// CNC/10 MessagesHandler/FB_ChannelError
FUNCTION_BLOCK FB_ChannelError
VAR_INPUT
	nChanIdx: INT;
END_VAR
VAR_OUTPUT
	Valid: BOOL := FALSE;
	/// Identification of channel error 
	ChErrorID: UDINT;
	/// Module name 
	ModuleName: STRING;
	/// Line in source file 
	Line: DINT;
	/// Multiple ID 
	MultipleID: DINT;
	/// Commandable function type 
	CmdFunctionType: DINT;
	/// Identification of the channel 
	ChannelID: DINT;
	/// Communication ID 
	CommuID: DINT;
	/// Cycle counter of CNC 
	CycleCounter: UDINT;
	/// Version name 
	VersionName: STRING;
	/// Remedy class of error 
	RemedyClass: DINT;
	/// Reaction class of error 
	ReactionClass: DINT;
	/// Body type of error 
	BodyType: UDINT;
	/// User message 
	UserMessage: STRING;
	/// Variables of error record body 
	BodyTypeEnum: UDINT;
	NcBlockNr: DINT := 0;
	ProgName: STRING := '';
	FileName: STRING := '';
	FileOffset: UDINT := 0;
	NcBlockOffset: DINT := 0;
	TokenOffset: DINT := 0;
	LogicalPathNr: DINT := 0;
	AddProgInfo: STRING := '';
	CommuMedium: DINT := 0;
	CommuType: UDINT := 0;
	CommuPartner: UDINT := 0;
	FileLine: UDINT := 0;
	ListType: DINT := 0;
	StructName: STRING := '';
	StrValue_1: STRING;
	StrValue_2: STRING;
	StrValue_3: STRING;
	StrValue_4: STRING;
	StrValue_5: STRING;
	MeaningValue_1: STRING;
	MeaningValue_2: STRING;
	MeaningValue_3: STRING;
	MeaningValue_4: STRING;
END_VAR
VAR
	/// Index of channel specific HLI area 	
	pMcError: POINTER TO MC_ERROR;
	pMcError2: POINTER TO MC_ERROR;
	SatzR: HLI_ERROR_SATZ;
	bInitialized: BOOL := FALSE;
	bClear: BOOL := FALSE;
	bUsed: ARRAY[0..CNC_EVENTS_MAXIDX] OF BOOL;
	bToCleanUp: ARRAY[0..CNC_EVENTS_MAXIDX] OF BOOL;
	LogEvent: ARRAY[0..CNC_EVENTS_MAXIDX] OF ADSLOGEVENT;
	FlankeQuit: ARRAY[0..CNC_EVENTS_MAXIDX] OF R_TRIG;
	pLog: POINTER TO ADSLOGEVENT;
	fmtStr: STRING;
	eventId: UDINT;
	i: UDINT;
	idx: UDINT := 0;
	maxWarnings: UINT;
	maxErrors: UINT;
	maxUserEvents: UINT;
	/// Gesamtzahl = Userevents und Errors 
	maxEvents: UINT;
	/// maximal index of an event 
	maxIdxEvents: UINT;
	countWarnings: UINT := 0;
	countErrors: UINT := 0;
	countUserEvents: UINT := 0;
	start_idx: UINT;
	stop_idx: UINT;
	paraPointerArray: ARRAY[0..31] OF POINTER TO UDINT;
	paraIndex: INT;
	pRumpfNcProg: POINTER TO HLI_RUMPF_NC_PROG;
	pRumpfNcProgLr: POINTER TO HLI_RUMPF_NC_PROG_LR;
	pRumpfMds: POINTER TO HLI_RUMPF_MDS;
	pRumpfKommu: POINTER TO HLI_RUMPF_KOMMU;
	pRumpfRamDisk: POINTER TO HLI_RUMPF_RAMDISK;
	pRumpfFile: POINTER TO HLI_RUMPF_FILE;
	pRumpfIntprFile: POINTER TO HLI_RUMPF_INTPR_FILE;
	pRumpfListeBinaer: POINTER TO HLI_RUMPF_LISTE_BINAER;
	pRumpfGcm: POINTER TO HLI_RUMPF_GCM;
	bTcComError: BOOL;
	bAxisErr: BOOL;
	nLogAxisId: DINT;
	
	// TC3 EventLogger
	fbADSRead : ADSREAD;
  	cnc_error_manager_mode_r : UDINT;
  	suppress_tc2_event_log_output : BOOL; 
	init : BOOL;
END_VAR
VAR CONSTANT
	XmlEventId_Rumpf: UDINT := 200;
	XmlEventId_RumpfNcProg: UDINT := 201;
	XmlEventId_RumpfNcProgLr: UDINT := 202;
	XmlEventId_RumpfMds: UDINT := 203;
	XmlEventId_RumpfKommu: UDINT := 204;
	XmlEventId_RumpfRamDisk: UDINT := 205;
	XmlEventId_RumpfFile: UDINT := 206;
	XmlEventId_RumpfIntprFile: UDINT := 207;
	XmlEventId_RumpfListeBinaer: UDINT := 208;
	XmlEventId_RumpfGcm: UDINT := 209;
	CNC_SOURCE_ID_BASE: UDINT := 551;
	CNC_USER_SOURCE_ID_BASE: UDINT := 651;
	MAX_CNC_ERRORS: UDINT := 49;
	MAX_CNC_USER_EVENTS: UDINT := 49;
	/// MAX_CNC_ERRORS + MAX_CNC_USER_EVENTS 
	MAX_CNC_EVENTS: UDINT := 98;
	/// MAX_CNC_EVENTS - 1 
	CNC_EVENTS_MAXIDX: UDINT := 97;
	ERR_BAHN_ONLINE_TRC_CALCULATION: UDINT := 50689;
	ERR_ID_REPORT_CNC_RESET: UDINT := 270076;
	ERR_ID_KIN_TRAFO_CONFIG: UDINT := 292030;
	ERR_ID_KIN_TRAFO_INIT: UDINT := 292031;
	ERR_ID_KIN_TRAFO_FORWARD: UDINT := 292032;
	ERR_ID_KIN_TRAFO_BACKWARD: UDINT := 292033;
END_VAR

(* ========================================================= *)
(*    FB: FB_ChannelError                               	 *)
(* --------------------------------------------------------- *)
(*   Desc: FB transfers CNC Errors to the Event Logger		 *)
(*   Author: ISG / TV                                        *)
(*   Date: 20.11.2018                                        *)
(*   Rev.: 1.6                                               *)
(*															 *)
(* ========================================================= *)

(* check for channel no *)
IF NOT HLI3_CheckChannelValid(nChannel := nChanIdx) THEN
	RETURN;
END_IF



// Check if TC3 EventLogger is active
fbADSRead(
	NETID:= '', 
	PORT:= 553, 
	IDXGRP:= 16#20101, 
	IDXOFFS:= 16#293, 
	LEN:= 4, 
	DESTADDR:= ADR(cnc_error_manager_mode_r ), 
	READ:= TRUE);
		
	IF NOT fbADSRead.BUSY THEN
		init := TRUE;
	END_IF
	
	IF NOT init THEN 
		RETURN;
	END_IF
			
	IF ((cnc_error_manager_mode_r AND 16#00080000) = 16#80000) THEN
		  suppress_tc2_event_log_output := TRUE;	
	END_IF


(* check for zero pointer *)
IF gpCh[nChanIdx] = 0 THEN
  RETURN;
END_IF

(* check for zero pointer, first channel is necessary for axis errors (Position controller errors) *)
IF gpCh[0] = 0 THEN
  RETURN;
END_IF

pMcError := ADR(gpCh[nChanIdx]^.mc_error);
SatzR    := pMcError^.satz_r;

IF bInitialized = FALSE THEN
  pMcError^.enable_w := TRUE;    (* enable control unit for error messages *) 
  bInitialized  := TRUE;
  maxErrors     := UDINT_TO_UINT(MAX_CNC_ERRORS / gNrCh);
  maxWarnings   := maxErrors / 5;
  maxUserEvents := UDINT_TO_UINT(MAX_CNC_USER_EVENTS / gNrCh);
  maxEvents     := maxUserEvents + maxErrors;

  maxIdxEvents := (maxEvents - 1);
  FOR i := 0 TO maxIdxEvents DO
    (* ----------------------------------------- *)
    (* initialize fixed elements of event        *)
    (* ----------------------------------------- *)
    pLog := ADR( LogEvent[i] );
    pLog^.NETID := '';      (* Local Computer *)
    pLog^.PORT:= 110;       (* Event Logger *)
    pLog^.TMOUT:= t#10s;
    pLog^.EventConfigData.Prio         := TCEVENTPRIO_IMPLICIT;
    pLog^.EventConfigData.ProgId       := 'TcEventFormatter.TcXmlFormatter';
    pLog^.EventConfigData.Flags        := TCEVENTFLAG_SRCID OR TCEVENTFLAG_LOG;
    pLog^.EventConfigData.SourceString := '';
    pLog^.EventConfigData.StreamType   := TCEVENTSTREAM_NORMAL;

    IF i < maxErrors THEN
      (* SourceID: 550 error texts, [ 551,  599] for single CNC error messages *)
      pLog^.EventConfigData.SourceId := CNC_SOURCE_ID_BASE + i + (DINT_TO_UINT(nChanIdx)*maxErrors);
    ELSE
      (* SourceID: 650 user error texts, [ 651,  699] for single CNC user error messages "ERROR[]" *)
      pLog^.EventConfigData.SourceId := CNC_USER_SOURCE_ID_BASE + i-maxErrors + (DINT_TO_UINT(nChanIdx)*maxUserEvents);
    END_IF

    FlankeQuit[i](CLK :=  pLog^.Quit);
  END_FOR
END_IF



(* -------------------------------------------------------------------------*)
(* test if events which have been reported shall be cleared again           *)
(* -------------------------------------------------------------------------*)
IF bClear THEN
  bClear := FALSE;
  countWarnings := 0;
  countErrors := 0;
  countUserEvents := 0;
  FOR i := 0 TO maxIdxEvents DO
    IF bToCleanup[i] = FALSE AND bUsed[i] THEN
      bToCleanup[i] := TRUE;
    END_IF
  END_FOR
END_IF


(* -------------------------------------------------------------------------*)
(* check for new error message                                              *)
(* -------------------------------------------------------------------------*)

(* Output for position controller errors is gpCh[0]^ *)
IF gpCh[0]^.mc_error.semaphor_rw THEN	
	SatzR := gpCh[0]^.mc_error.satz_r;		
	bAxisErr := TRUE;				
END_IF

IF (pMcError^.semaphor_rw  OR bAxisErr)  THEN

 	IF  SatzR.kopf.cnc_channel > 0 THEN 
  		IF (SatzR.kopf.cnc_channel-1 <> INT_TO_UINT(nChanIdx)) THEN	  
			bAxisErr := FALSE;		
    	RETURN;
	END_IF
  END_IF
  
  (* Initialize output variables that depend on error body type *)
  NcBlockNr      := 0;
  ProgName       := '';
  FileName       := '';
  FileOffset     := 0;
  NcBlockOffset  := 0;
  TokenOffset    := 0;
  LogicalPathNr  := 0;
  AddProgInfo    := '';

  CommuMedium    := 0;
  CommuType      := 0;
  CommuPartner   := 0;

  FileLine       := 0;
  ListType       := 0;
  StructName     := '';

  StrValue_1     := '';
  StrValue_2     := '';
  StrValue_3     := '';
  StrValue_4     := '';
  StrValue_5     := '';

  MeaningValue_1 := '';
  MeaningValue_2 := '';
  MeaningValue_3 := '';
  MeaningValue_4 := '';
  
  nLogAxisId   := 0;


  eventId := SatzR.kopf.error_id;

  (*------------------------------------------------------------------*)
  (* automatic clear old events if CNC reports reset                  *)
  (*------------------------------------------------------------------*)
  IF eventId = ERR_ID_REPORT_CNC_RESET THEN
	  	IF bAxisErr THEN 
    		gpCh[0]^.mc_error.semaphor_rw := FALSE;
			bAxisErr := FALSE;
		ELSE
			pMcError^.semaphor_rw := FALSE;		
		END_IF
	
    bClear := TRUE;
    RETURN;
  END_IF

  
  (*------------------------------------------------------------------*)
  (* TcCom: kinematic transformation, map util_error_id to error_id   *)
  (*------------------------------------------------------------------*)
  IF    eventId = ERR_ID_KIN_TRAFO_CONFIG
     OR eventId = ERR_ID_KIN_TRAFO_INIT  
     OR eventId = ERR_ID_KIN_TRAFO_FORWARD
     OR eventId = ERR_ID_KIN_TRAFO_BACKWARD
   OR eventId = ERR_BAHN_ONLINE_TRC_CALCULATION
  THEN
    eventId := SatzR.kopf.util_error_id;
    bTcComError := TRUE;
  ELSE
    bTcComError := FALSE;
  END_IF
   

  (*-------------------------------*)
  (* search unused event           *)
  (*-------------------------------*)
  IF eventId <= 1000 OR bTcComError THEN
    countUserEvents := countUserEvents + 1;
    start_idx       := maxErrors;
    stop_idx        := maxErrors + maxUserEvents - 1;
  ELSE
    (*------------------------------------------------------------------*)
    (* check maximum number of active warnings                          *)
    (*------------------------------------------------------------------*)
    IF SatzR.kopf.behebungs_klasse < 2 THEN
      IF countWarnings > maxWarnings THEN
		  IF (bAxisErr) THEN
			  	gpCh[0]^.mc_error.semaphor_rw := FALSE;
				bAxisErr := FALSE;
		  ELSE	
				pMcError^.semaphor_rw := FALSE;	  
		  END_IF
        
        RETURN;  (* dismiss further warning *)
      END_IF
      countWarnings:= countWarnings + 1;
    END_IF

    countErrors := countErrors + 1;
    start_idx   := 0;
    stop_idx    := maxErrors - 1;
  END_IF

  FOR i := start_idx TO stop_idx DO
    IF bUsed[i] = FALSE THEN
      EXIT;
    END_IF
  END_FOR

  IF i > stop_idx THEN
    (*------------------------------------------------------------------*)
    (* overflow -> dismiss actual message, wait for reset               *)
    (*------------------------------------------------------------------*)
	IF (bAxisErr) THEN
		gpCh[0]^.mc_error.semaphor_rw := FALSE;
		bAxisErr := FALSE;
	ELSE	
		pMcError^.semaphor_rw := FALSE;	  
	END_IF	
    RETURN;
  END_IF
  idx := i;


  bUsed[idx] := TRUE;
  pLog := ADR( LogEvent[idx] );

  (* Initialisierungen fuer jeden Aufruf *)
  paraIndex := 0;

  (*
    TCEVENTCLASS_NONE        := 0,  No class
    TCEVENTCLASS_MAINTENANCE := 1,  Maintenance hint
    TCEVENTCLASS_MESSAGE     := 2,  Message
    TCEVENTCLASS_HINT        := 3,  Hint
    TCEVENTCLASS_STATEINFO   := 4,  State information
    TCEVENTCLASS_INSTRUCTION := 5,  Instruction
    TCEVENTCLASS_WARNING     := 6,  Warning
    TCEVENTCLASS_ALARM       := 7,  Alarm
    TCEVENTCLASS_PARAMERROR
  *)

  IF SatzR.kopf.behebungs_klasse < 2 THEN
    pLog^.EventConfigData.Class := TCEVENTCLASS_WARNING;
    pLog^.EventConfigData.bQuitRequired := FALSE;  (* Hasn't to acknowledge the event *)
  ELSE
    pLog^.EventConfigData.bQuitRequired := TRUE;  (* Has to acknowledge the event *)
    IF SatzR.kopf.behebungs_klasse < 7 THEN
      pLog^.EventConfigData.Class := TCEVENTCLASS_ALARM;
    ELSE
      pLog^.EventConfigData.Class := TCEVENTCLASS_PARAMERROR;
    END_IF
  END_IF
  pLog^.EventConfigData.Id := XmlEventId_Rumpf;

  (*------------------------------------------------------------------*)
  (* parameters 1 - 13 are content independent                        *)
  (*------------------------------------------------------------------*)
  fmtStr := '%d%d%d%d%s%d%d%d%d%d%s%d%s';  (* a string *)

  (* If ChErrorID has a link to a sub string (other EventId and SourceId)  *)
  (* a string is build of following syntax: '[SxEy]' with x as SourceId and y as EventId *)
  (* in TcCncError.xml x alsways has value 2 and y is the ChErrorID of the CNC *)
  (* ----------------------------------------------------*)
  (* User specific error message                         *)
  (* ----------------------------------------------------*)
  IF eventId <= 1000 OR bTcComError THEN
    UserMessage   := '[S650E'; (* sub string from SourceId 550 (see TcCncUserEvents.xml) and EventId 'eventId' *)
  ELSE
    UserMessage   := '[S550E'; (* sub string from SourceId 2 (see TcCncError.xml) and EventId 'eventId' *)
  END_IF
  UserMessage     := CONCAT(UserMessage, UDINT_TO_STRING(eventId));
  UserMessage     := CONCAT(UserMessage, ']');

  ChErrorID       := eventId;
  ChannelID       := SatzR.kopf.cnc_channel;
  RemedyClass     := SatzR.kopf.behebungs_klasse;
  ReactionClass   := SatzR.kopf.reaktions_klasse;
  ModuleName      := SatzR.kopf.modul_name.zeichen;
  Line            := SatzR.kopf.line;
  MultipleID      := SatzR.kopf.multiple_id;
  CmdFunctionType := SatzR.kopf.bf_type;

  CommuID         := SatzR.kopf.kommu_id;
  CycleCounter    := SatzR.kopf.fb_zeitangabe.zykl_counter;
  VersionName     := SatzR.kopf.version_name.zeichen;
  BodyType        := SatzR.kopf.rumpf_typ;

  paraPointerArray[paraIndex] := ADR(ChErrorID);
  paraIndex := paraIndex + 1;
  paraPointerArray[paraIndex] := ADR(ChannelID);
  paraIndex := paraIndex + 1;
  paraPointerArray[paraIndex] := ADR(RemedyClass);
  paraIndex := paraIndex + 1;
  paraPointerArray[paraIndex] := ADR(ReactionClass);
  paraIndex := paraIndex + 1;
  paraPointerArray[paraIndex] := ADR(ModuleName);
  paraIndex := paraIndex + 1;
  paraPointerArray[paraIndex] := ADR(Line);
  paraIndex := paraIndex + 1;
  paraPointerArray[paraIndex] := ADR(MultipleID);
  paraIndex := paraIndex + 1;
  paraPointerArray[paraIndex] := ADR(CmdFunctionType);
  paraIndex := paraIndex + 1;
  paraPointerArray[paraIndex] := ADR(CommuID);
  paraIndex := paraIndex + 1;
  paraPointerArray[paraIndex] := ADR(CycleCounter);
  paraIndex := paraIndex + 1;
  paraPointerArray[paraIndex] := ADR(VersionName);
  paraIndex := paraIndex + 1;
  paraPointerArray[paraIndex] := ADR(BodyType);
  paraIndex := paraIndex + 1;
  paraPointerArray[paraIndex] := ADR(UserMessage);
  paraIndex := paraIndex + 1;


  (*------------------------------------------------------------------------*)
  (* Append values and meaning of values.                                   *)
  (*------------------------------------------------------------------------*)
  
  StrValue_1 := CNCErrorParameterToString(SatzR.rumpf.wert_1, 1);
  StrValue_2 := CNCErrorParameterToString(SatzR.rumpf.wert_2, 2);
  StrValue_3 := CNCErrorParameterToString(SatzR.rumpf.wert_3, 3);
  StrValue_4 := CNCErrorParameterToString(SatzR.rumpf.wert_4, 4);
  StrValue_5 := CNCErrorParameterToString(SatzR.rumpf.wert_5, 5);  
   
  CNCErrorGetLogAxisId(SatzR.rumpf.wert_1,nLogAxisId);
  CNCErrorGetLogAxisId(SatzR.rumpf.wert_2,nLogAxisId);
  CNCErrorGetLogAxisId(SatzR.rumpf.wert_3,nLogAxisId);
  CNCErrorGetLogAxisId(SatzR.rumpf.wert_4,nLogAxisId);
  CNCErrorGetLogAxisId(SatzR.rumpf.wert_5,nLogAxisId);
  
  CNCSystem.LogAxisNo[nLogAxisId].nCNCErrorID :=  ChErrorID;
     
  paraPointerArray[paraIndex] := ADR(StrValue_1);
  paraIndex := paraIndex + 1;
  paraPointerArray[paraIndex] := ADR(StrValue_2);
  paraIndex := paraIndex + 1;
  paraPointerArray[paraIndex] := ADR(StrValue_3);
  paraIndex := paraIndex + 1;
  paraPointerArray[paraIndex] := ADR(StrValue_4);
  paraIndex := paraIndex + 1;
  paraPointerArray[paraIndex] := ADR(StrValue_5);
  paraIndex := paraIndex + 1;

  fmtStr := CONCAT(fmtStr, '%s%s%s%s%s');

  MeaningValue_1 := WertToString(SatzR.rumpf.kennung_1, 1);
  MeaningValue_2 := WertToString(SatzR.rumpf.kennung_2, 2);
  MeaningValue_3 := WertToString(SatzR.rumpf.kennung_3, 3);
  MeaningValue_4 := WertToString(SatzR.rumpf.kennung_4, 4);

  paraPointerArray[paraIndex] := ADR(MeaningValue_1);
  paraIndex := paraIndex + 1;
  paraPointerArray[paraIndex] := ADR(MeaningValue_2);
  paraIndex := paraIndex + 1;
  paraPointerArray[paraIndex] := ADR(MeaningValue_3);
  paraIndex := paraIndex + 1;
  paraPointerArray[paraIndex] := ADR(MeaningValue_4);
  paraIndex := paraIndex + 1;

  fmtStr := CONCAT(fmtStr, '%s%s%s%s');



  BodyTypeEnum := SatzR.kopf.rumpf_typ;

  (*-------------------------------------------------------------------------*)
  (*       HLI_RUMPF_TYP_NC_PROG                                             *)
  (*-------------------------------------------------------------------------*)
  IF BodyTypeEnum = HLI_RUMPF_TYP_NC_PROG THEN
    pLog^.EventConfigData.Id := XmlEventId_RumpfNcProg;

    pRumpfNcProg := ADR(SatzR.rumpf.maske);

    (* Assign error body data to output variables *)
    NcBlockNr     := pRumpfNcProg^.satz_nr;
    ProgName      := pRumpfNcProg^.prog_name.zeichen;
    FileName      := pRumpfNcProg^.file_name.zeichen;
    FileOffset    := pRumpfNcProg^.fileoffset;
    NcBlockOffset := pRumpfNcProg^.satzoffset;
    TokenOffset   := pRumpfNcProg^.tokenoffset;
    LogicalPathNr := pRumpfNcProg^.log_pfad_nr;
    AddProgInfo   := ''; //  pRumpfNcProg^.add_prog_info.zeichen;

    (* Assign address of data to parameter array of the event *)
    paraPointerArray[paraIndex] := ADR(NcBlockNr);
    paraIndex := paraIndex + 1;
    paraPointerArray[paraIndex] := ADR(ProgName);
    paraIndex := paraIndex + 1;
    paraPointerArray[paraIndex] := ADR(FileName);
    paraIndex := paraIndex + 1;
    paraPointerArray[paraIndex] := ADR(FileOffset);
    paraIndex := paraIndex + 1;
    paraPointerArray[paraIndex] := ADR(NcBlockOffset);
    paraIndex := paraIndex + 1;
    paraPointerArray[paraIndex] := ADR(TokenOffset);
    paraIndex := paraIndex + 1;
    paraPointerArray[paraIndex] := ADR(LogicalPathNr);
    paraIndex := paraIndex + 1;
    paraPointerArray[paraIndex] := ADR(AddProgInfo);
    paraIndex := paraIndex + 1;

    (* Add format string for error messages out of NC programs *)
    fmtStr := CONCAT(fmtStr, '%d%s%s%d%d%d%d%s');
  (*-------------------------------------------------------------------------*)
  (*       HLI_RUMPF_TYP_NC_PROG_LR                                          *)
  (*-------------------------------------------------------------------------*)
  ELSIF BodyTypeEnum = HLI_RUMPF_TYP_NC_PROG_LR THEN
    pLog^.EventConfigData.Id := XmlEventId_RumpfNcProgLR;

    pRumpfNcProgLr := ADR(SatzR.rumpf.maske);

    LogicalPathNr  := pRumpfNcProgLr^.log_pfad_nr;
    ProgName       := pRumpfNcProgLr^.prog_name.zeichen;
    FileName       := pRumpfNcProgLr^.file_name.zeichen;
    NcBlockNr      := pRumpfNcProgLr^.satz_nr;
    AddProgInfo    := ''; //pRumpfNcProgLr^.add_prog_info.zeichen;

    paraPointerArray[paraIndex] := ADR(NcBlockNr);
    paraIndex := paraIndex + 1;
    paraPointerArray[paraIndex] := ADR(ProgName);
    paraIndex := paraIndex + 1;
    paraPointerArray[paraIndex] := ADR(FileName);
    paraIndex := paraIndex + 1;
    paraPointerArray[paraIndex] := ADR(LogicalPathNr);
    paraIndex := paraIndex + 1;
    paraPointerArray[paraIndex] := ADR(AddProgInfo);
    paraIndex := paraIndex + 1;

    fmtStr := CONCAT(fmtStr, '%d%s%s%d%s');
  (*-------------------------------------------------------------------------*)
  (*       HLI_RUMPF_TYP_MDS                                                 *)
  (*-------------------------------------------------------------------------*)
  ELSIF BodyTypeEnum = HLI_RUMPF_TYP_MDS THEN
    pLog^.EventConfigData.Id := XmlEventId_RumpfMds;

    pRumpfMds     := ADR(SatzR.rumpf.maske);

    LogicalPathNr := pRumpfMds^.listen_typ;
    ProgName      := pRumpfMds^.strukt_name.zeichen;

    paraPointerArray[paraIndex] := ADR(LogicalPathNr);
    paraIndex := paraIndex + 1;
    paraPointerArray[paraIndex] := ADR(ProgName);
    paraIndex := paraIndex + 1;

    fmtStr := CONCAT(fmtStr, '%d%s');
  (*-------------------------------------------------------------------------*)
  (*       HLI_RUMPF_TYP_KOMMU                                               *)
  (*-------------------------------------------------------------------------*)
  ELSIF BodyTypeEnum = HLI_RUMPF_TYP_KOMMU THEN
    pLog^.EventConfigData.Id := XmlEventId_RumpfKommu;

    pRumpfKommu  := ADR(SatzR.rumpf.maske);

    CommuMedium  := pRumpfKommu^.Medium;
    CommuType    := pRumpfKommu^.Typ;
    CommuPartner := pRumpfKommu^.Partner;

    paraPointerArray[paraIndex] := ADR(CommuMedium);
    paraIndex := paraIndex + 1;
    paraPointerArray[paraIndex] := ADR(CommuType);
    paraIndex := paraIndex + 1;
    paraPointerArray[paraIndex] := ADR(CommuPartner);
    paraIndex := paraIndex + 1;

    fmtStr := CONCAT(fmtStr, '%d%d%d');
  (*-------------------------------------------------------------------------*)
  (*       HLI_RUMPF_TYP_RAMDISK                                             *)
  (*-------------------------------------------------------------------------*)
  ELSIF BodyTypeEnum = HLI_RUMPF_TYP_RAMDISK THEN
    pLog^.EventConfigData.Id := XmlEventId_RumpfRamDisk;

    pRumpfRamDisk := ADR(SatzR.rumpf.maske);

    CommuMedium   := pRumpfRamDisk^.medium;
    CommuType     := pRumpfRamDisk^.typ;
    CommuPartner  := pRumpfRamDisk^.partner;
    FileName      := pRumpfRamDisk^.file_name.zeichen;
    FileOffset    := pRumpfRamDisk^.fileoffset;

    paraPointerArray[paraIndex] := ADR(CommuMedium);
    paraIndex := paraIndex + 1;
    paraPointerArray[paraIndex] := ADR(CommuType);
    paraIndex := paraIndex + 1;
    paraPointerArray[paraIndex] := ADR(CommuPartner);
    paraIndex := paraIndex + 1;
    paraPointerArray[paraIndex] := ADR(FileName);
    paraIndex := paraIndex + 1;
    paraPointerArray[paraIndex] := ADR(FileOffset);
    paraIndex := paraIndex + 1;

    fmtStr := CONCAT(fmtStr, '%d%d%d%s%d');
  (*-------------------------------------------------------------------------*)
  (*       HLI_RUMPF_TYP_FILE                                                *)
  (*-------------------------------------------------------------------------*)
  ELSIF BodyTypeEnum = HLI_RUMPF_TYP_FILE THEN
    pLog^.EventConfigData.Id := XmlEventId_RumpfFile;

    pRumpfFile := ADR(SatzR.rumpf.maske);

    FileName   := pRumpfFile^.file_name.zeichen;
    FileOffset := pRumpfFile^.fileoffset;

    paraPointerArray[paraIndex] := ADR(FileName);
    paraIndex := paraIndex + 1;
    paraPointerArray[paraIndex] := ADR(FileOffset);
    paraIndex := paraIndex + 1;

    fmtStr := CONCAT(fmtStr, '%s%d');
  (*-------------------------------------------------------------------------*)
  (*       HLI_RUMPF_TYP_INTPR_FILE                                          *)
  (*-------------------------------------------------------------------------*)
  ELSIF BodyTypeEnum = HLI_RUMPF_TYP_INTPR_FILE THEN
    pLog^.EventConfigData.Id := XmlEventId_RumpfIntprFile;

    pRumpfIntprFile := ADR(SatzR.rumpf.maske);

    FileName   := pRumpfIntprFile^.file_name.zeichen;
    FileOffset := pRumpfIntprFile^.fileoffset;
    FileLine   := pRumpfIntprFile^.file_line_number;
    ListType   := pRumpfIntprFile^.listen_typ;
    StructName := pRumpfIntprFile^.strukt_name.zeichen;

    paraPointerArray[paraIndex] := ADR(FileName);
    paraIndex := paraIndex + 1;
    paraPointerArray[paraIndex] := ADR(FileOffset);
    paraIndex := paraIndex + 1;
    paraPointerArray[paraIndex] := ADR(FileLine);
    paraIndex := paraIndex + 1;
    paraPointerArray[paraIndex] := ADR(ListType);
    paraIndex := paraIndex + 1;
    paraPointerArray[paraIndex] := ADR(StructName);
    paraIndex := paraIndex + 1;

    fmtStr := CONCAT(fmtStr, '%s%d%d%d%s');
  (*-------------------------------------------------------------------------*)
  (*       HLI_RUMPF_TYP_LISTE_BINAER                                        *)
  (*-------------------------------------------------------------------------*)
  ELSIF BodyTypeEnum = HLI_RUMPF_TYP_LISTE_BINAER THEN
    pLog^.EventConfigData.Id := XmlEventId_RumpfListeBinaer;

    pRumpfListeBinaer := ADR(SatzR.rumpf.maske);

    StructName:=pRumpfListeBinaer^.strukt_name.zeichen;

    paraPointerArray[paraIndex] := ADR(StructName);
    paraIndex := paraIndex + 1;

    fmtStr := CONCAT(fmtStr, '%s');
  (*-------------------------------------------------------------------------*)
  (*       HLI_RUMPF_TYP_GCM                                                 *)
  (*-------------------------------------------------------------------------*)
  ELSIF BodyTypeEnum = HLI_RUMPF_TYP_GCM THEN
    pLog^.EventConfigData.Id := XmlEventId_RumpfGcm;

    pRumpfGcm := ADR(SatzR.Rumpf.Maske);

    ProgName:=pRumpfGcm^.Token.zeichen;
    FileName:=pRumpfGcm^.FileName.zeichen;

    paraPointerArray[paraIndex] := ADR(ProgName);
    paraIndex := paraIndex + 1;
    paraPointerArray[paraIndex] := ADR(FileName);
    paraIndex := paraIndex + 1;

    fmtStr := CONCAT(fmtStr, '%s%s');
  END_IF
  
  
   // IF TC3 EventLogger : no output to event logger needed  	   
   IF suppress_tc2_event_log_output THEN
	   IF (bAxisErr) THEN
			gpCh[0]^.mc_error.semaphor_rw := FALSE;
			bAxisErr := FALSE;
		ELSE	
			pMcError^.semaphor_rw := FALSE;	  
		END_IF
		
	   RETURN;   
   END_IF
  
  
  (*------------------------------------------------------------------------*)
  (* Set values at input pins of FB                                         *)
  (*------------------------------------------------------------------------*)
  pLog^.EventDataAddress:= ADR(paraPointerArray);
  pLog^.EventDataLength:= 0;
  pLog^.fbCleanUp  := FALSE;
  pLog^.EventQuit  := FALSE;

  pLog^.EventConfigData.DataFormatStrAddress := ADR(fmtStr);

  (*------------------------------------------------------------------------*)
  (* report error message to event logger                                   *)
  (*------------------------------------------------------------------------*)
  pLog^(Event := TRUE);

  (* Notify at output that a error essage occurred *)
  Valid := TRUE;

  (* Acknowledge error message *)
 	IF (bAxisErr) THEN
		gpCh[0]^.mc_error.semaphor_rw := FALSE;
		bAxisErr := FALSE;
	ELSE	
		pMcError^.semaphor_rw := FALSE;	  
	END_IF
ELSE
  Valid := FALSE;
END_IF

(* by default : no error message is present, first search for error messages *)
FOR i := 0 TO maxIdxEvents DO
  (*-------------------------------------------------------------------------*)
  (*       clear event                                                       *)
  (*-------------------------------------------------------------------------*)
  IF bToCleanup[i] THEN
    pLog := ADR( LogEvent[i] );
    pLog^();

    IF pLog^.EventState=TCEVENTSTATE_SIGNALED THEN
      pLog^( Event:=FALSE);
    ELSIF pLog^.EventState=TCEVENTSTATE_RESET THEN
      pLog^( EventQuit:= TRUE);
    ELSIF pLog^.EventState=TCEVENTSTATE_CONFIRMED OR pLog^.EventState=TCEVENTSTATE_INVALID THEN
      (*pLog^( FbCleanup:= TRUE); bugfix 12.7.2005*)
      bUsed[i]     := FALSE;
      bToCleanup[i] := FALSE;
    END_IF;
  (*-------------------------------------------------------------------------*)
  (*       report event                                                      *)
  (*-------------------------------------------------------------------------*)
  ELSIF bUsed[i] THEN
    pLog := ADR( LogEvent[i] );
    pLog^();

    (* IF pLog^.EventConfigData.bQuitRequired = FALSE THEN
      FlankeQuit[i](CLK :=  pLog^.Quit);
      IF FlankeQuit[i].Q = TRUE THEN
        bUsed[i] := FALSE;
        QuitCount := QuitCount + 1;
      END_IF
    END_IF*)
  END_IF
END_FOR

END_FUNCTION_BLOCK

// CNC/11 Util/F_GRAYCODE_TO_UINT
FUNCTION F_GRAYCODE_TO_UINT : UINT
VAR_INPUT
	byGraycodeSwitches	: BYTE;
END_VAR
VAR
	nLoopCount				: INT;
	byResult					: BYTE;
	bySwitches				: BYTE;
END_VAR

bySwitches			:= byGraycodeSwitches;
byResult				:= 0;

FOR nLoopCount := 0 TO 31 DO
	byResult 		:= byResult XOR bySwitches;
	bySwitches		:= SHR(bySwitches, 1);
END_FOR

F_GRAYCODE_TO_UINT	:= BYTE_TO_UINT(byResult);

END_FUNCTION

// CNC/11 Util/FB_ActivateVolCompList
FUNCTION_BLOCK FB_ActivateVolCompList
VAR_INPUT
	bExecute			: BOOL;
	strPathParamList 	: STRING(256);
	nIndex				: UINT;
	tTimeout			: TIME := T#10S;
END_VAR
VAR_OUTPUT
	bBusy			: 	BOOL;
	bError			:	BOOL;
	nErrID			:	UDINT;
END_VAR
VAR
	iState 			:  UINT;
	fbOnTrigger		:  R_TRIG;
	fbAdsWrite		:  ADSWRITE;
END_VAR

(* ========================================================= *)
(*     FB: FB_WriteVolCompParam                              *)
(* --------------------------------------------------------- *)
(*   Desc:  Write Volumetric Compensation Parameter to CNC   *)
(*   Author: TV				                                 *)
(*   Date: 2018.04.27                                        *)
(*   Rev.: 1.0                                               *)
(* ==========================================================*)

fbOnTrigger(CLK:= bExecute);

IF fbOnTrigger.Q THEN
	iState := 10;
	nErrID := 0;
	bError := 0;
	bBusy := TRUE;
	fbAdsWrite(WRITE := FALSE);
END_IF



CASE iState OF

0:
	bBusy := FALSE;
	
10: // Write Index
	fbAdsWrite( Port := 553, IdxGrp := 16#20101, IdxOffs := (16#27D), LEN := SIZEOF(nIndex), SrcAddr := ADR(nIndex), WRITE := TRUE);
	iState := 20;
	
20:	IF NOT fbAdsWrite.Busy THEN
			IF fbAdsWrite.Err THEN
				bError := fbAdsWrite.Err;
				nErrID :=fbAdsWrite.ERRID;
				iState := 0;
			ELSE
				fbAdsWrite(WRITE := FALSE);
				iState := 30;
			END_IF
		END_IF
		
		
30:
	(* Set Parameter List file *)
    FbAdsWrite( Port := 553, IdxGrp := 16#20101, IdxOffs := (16#27C), LEN := SIZEOF(strPathParamList), SrcAddr := ADR(strPathParamList), WRITE := TRUE);
	iState := 40;
	
40:
		IF NOT fbAdsWrite.Busy THEN
			IF fbAdsWrite.Err THEN
				bError := fbAdsWrite.Err;
				nErrID :=fbAdsWrite.ERRID;
				iState := 0;
			ELSE
				fbAdsWrite(WRITE := FALSE);
				iState := 0;
			END_IF
		END_IF


END_CASE

FbAdsWrite();

END_FUNCTION_BLOCK

// CNC/11 Util/FB_CNCWriteParameter
///*********************************************************************************************************
///NAME.......................:		FB_CNCWriteParameter
///DATUM....................:		08.12.2017, 27.06.2019
///AUTOR....................:		Thomas Voß, Michael Balsfulland
///VERSION................:			1.5
///
///Description.: 	The function block allows to write cnc parameters to the CNC kernel.					
///**********************************************************************************************************
FUNCTION_BLOCK FB_CNCWriteParameter
VAR_INPUT
	/// Channel Id	
	nLogChannelID : UINT;
	/// log. Axis Id  
	nLogAxisId: UINT;
	bExecute: BOOL;
	/// numbers of parameters 
	nNumParameters: INT;
	/// Parameter type
	eParameterType: E_CNCParameterTypes;
	/// Windows temp file for sub lists
	strTempPath: STRING;
	stParameter: ARRAY[0..199] OF ST_CNCParameter;
END_VAR
VAR_OUTPUT
	bBusy: BOOL;
	bError: BOOL;
	nErrorID: INT;
END_VAR

VAR
	fbOnTrigger: R_TRIG;
	Step: UDINT;
	FbAdsWrite: ADSWRITE;
	strParameterLine: STRING(255);
	strFileName: STRING(255);
	strHeader: STRING(255);
	TimeOut: TON;
	m: DINT;
	/// Text To File 
	fbFileOpen: FB_FileOpen;
	fbFileRead: FB_FileRead;
	fbFilePuts: FB_FilePuts;
	fbFileClose: FB_FileClose;
	hFileOutput: UINT := 0;
END_VAR
VAR CONSTANT
	nMaxParameters: INT := 200;
	/// Ads Interface 
	nAdsPortNumber: UINT := 553;
	nAdsIndexGroup: UDINT := 16#20100;
	nAdsIndexGroupAxisParameter: UDINT := 16#20200;
	nAdsIndexOffsetlogAxisNumber: UDINT := 16#37;
	nAdsIndexOffsetChannelParameter: UDINT := 16#34;	
	nAdsIndexOffsetAxisParameter: UDINT := 16#18;
	nAdsIndexOffsetZeroOffsets: UDINT := 16#2E;
	nAdsIndexOffsetToolParameter: UDINT := 16#30;
	nAdsIndexOffsetClampPosition: UDINT := 16#32;
	nAdsIndexOffsetCompensationTable: UDINT := 16#39;
	/// Time Out Error 
	ErrID_1: INT := 1;
	/// Fehler beim Öffnen der Parameterdatei 
	ErrID_2: INT := 2;
	/// ADS - Fehler : Vorgabe Achs ID 
	ErrID_3: INT := 3;
	/// ADS - Fehler : Aktivierung der Parameterliste 
	ErrID_4: INT := 4;
	/// Invalid   CNC Parameter Type 
	ErrID_5: INT := 5;
	/// Invalid   Axis Number  
	ErrID_6: INT := 6;
	/// Invalid   Channel Number  
	ErrID_7: INT := 7;
	/// Invalid   Number  of Parameters 
	ErrID_8: INT := 8;
	/// File Error 
	ErrID_9: INT := 9;
	/// Invalid Channel State 
	ErrID_10: INT := 10;
END_VAR



fbOnTrigger(CLK:= bExecute);

IF fbOnTrigger.Q THEN
	Step 	:= 10;
	nErrorID 	:= 0;
	bError	 := 0;
	bBusy := TRUE;
END_IF

CASE Step OF
0:
	bBusy := FALSE;

10: (* check input parameters *)
	IF (nNumParameters < 1 OR nNumParameters > nMaxParameters) THEN
		nErrorID 	:= ErrID_8;
		Step := 999;
	ELSE
		CASE eParameterType OF
				
			CNC_AxisParameter:
				IF (nLogAxisId <= 0  OR nLogAxisId > MAX_SYS_LOG_AXIS_INDEX) THEN
					nErrorID 	:= ErrID_6;
					Step := 999;
	
				ELSIF (nLogChannelID <= 0 OR nLogChannelID	 > nLogChannelID	) THEN
					nErrorID 	:= ErrID_7;
					Step := 999;
				ELSE
					Step := 12;
				END_IF

			CNC_ChannelParameter:
				IF (nLogChannelID <= 0 OR nLogChannelID > nLogChannelID) THEN
					nErrorID 	:= ErrID_7;
					Step := 999;
				ELSE
					Step := 12;
				END_IF

			CNC_ToolParameter:
				IF (nLogChannelID <= 0 OR nLogChannelID > nLogChannelID) THEN
					nErrorID 	:= ErrID_7;
					Step := 999;
				ELSE
					Step := 12;
				END_IF
	
			CNC_ClampPosition:
				IF (nLogChannelID <= 0 OR nLogChannelID > nLogChannelID) THEN
					nErrorID 	:= ErrID_7;
					Step := 999;
				ELSE
					Step := 12;
				END_IF
	
			CNC_ZeroOffsets:
				IF (nLogChannelID <= 0 OR nLogChannelID > nLogChannelID) THEN
					nErrorID 	:= ErrID_7;
					Step := 999;
				ELSE
					Step := 12;
				END_IF
		END_CASE
	END_IF

	fbFileOpen.bExecute := FALSE;
	
	// Check Channel State
	IF (CNCSystem.LogChannelNo[nLogChannelID].nHliChannelIdx <> -1) THEN
		;    // 2019.06.27 removed because it is possible to write parameter in any state  	
//		IF (cncSystem.Channel[CNCSystem.LogChannelNo[nLogChannelID].nHliChannelIdx].ActState <> HLI_IMCM_PROCESS_SELECTED AND 
//			cncSystem.Channel[CNCSystem.LogChannelNo[nLogChannelID].nHliChannelIdx].ActState <> HLI_IMCM_PROCESS_READY) THEN
//			nErrorID 	:= ErrID_10;
//			Step := 999;
//		END_IF				
	ELSE
			nErrorID 	:= ErrID_7;
			Step := 999;		
	END_IF			

12:	(* create file name and list file header  *)
	strHeader := '';

	CASE eParameterType OF

		CNC_AxisParameter:
			strFileName := CONCAT(strTempPath, '\axis');
			strFileName := CONCAT(strFileName, UINT_TO_STRING(nLogAxisId));
			strFileName := CONCAT(strFileName, '.lis');

			strHeader := 'kopf.achs_nr ';
			strHeader := CONCAT(strHeader, UINT_TO_STRING(nLogAxisId));
			Step := 15;
		CNC_ChannelParameter:
			strFileName := CONCAT(strTempPath, '\channel');			
			strFileName := CONCAT(strFileName, UINT_TO_STRING(nLogChannelID));
			strFileName := CONCAT(strFileName, '.lis');
			Step := 15;
		CNC_ToolParameter:			
			strFileName := CONCAT(strTempPath, '\ToolCh');
			strFileName := CONCAT(strFileName, UINT_TO_STRING(nLogChannelID));
			strFileName := CONCAT(strFileName, '.lis');
			Step := 15;
		CNC_ClampPosition:
			strFileName := CONCAT(strTempPath, '\ClampPosCh');			
			strFileName := CONCAT(strFileName, UINT_TO_STRING(nLogChannelID));
			strFileName := CONCAT(strFileName, '.lis');
			Step := 15;
		CNC_ZeroOffsets:			
			strFileName := CONCAT(strTempPath, '\ZeroOffsetsChh');
			strFileName := CONCAT(strFileName, UINT_TO_STRING(nLogChannelID));
			strFileName := CONCAT(strFileName, '.lis');
			Step := 15;
		ELSE
			nErrorID 	:= ErrID_5;
			Step := 999;
	END_CASE

15:	(* write file to destination folder *)
	fbFileOpen.sNetId := '';
	fbFileOpen.sPathName := strFileName;
	fbFileOpen.nMode := FOPEN_MODEWRITE OR FOPEN_MODETEXT;
	fbFileOpen.ePath := PATH_GENERIC;
	fbFileOpen.tTimeout := t#1s;
	fbFileOpen.bExecute := TRUE;
	Step := 16;

16:
	IF ( NOT fbFileOpen.bBusy ) THEN
		IF ( fbFileOpen.bError ) THEN
			nErrorID  :=ErrID_9 ;
			bError := TRUE;
			Step := 999;
		ELSE
			hFileOutput := fbFileOpen.hFile;
			fbFilePuts.bExecute:= FALSE;
			Step := 17;
		END_IF
	END_IF


17: (* Write Header File *)
	fbFilePuts.sNetId:='';
	fbFilePuts.hFile:=hFileOutput;
	fbFilePuts.bExecute:=TRUE;
	fbFilePuts.tTimeout:=t#10s;
	fbFilePuts.sLine :=strHeader;
	Step := 18;

18:
	IF ( NOT fbFilePuts.bBusy ) THEN
		IF ( fbFilePuts.bError ) THEN
			 nErrorID  :=ErrID_9 ;
			bError := TRUE;
			Step := 999;
		ELSE
			fbFilePuts.bExecute:= FALSE;
			m := 0;
			Step := 19;
		END_IF
	END_IF


19:	(* Write Parameter lines *)
		strParameterLine :=  CONCAT('$N',stParameter[m].strName);
		strParameterLine :=  CONCAT(strParameterLine,'   ');
		strParameterLine := CONCAT(strParameterLine, stParameter[m].strValue);
		fbFilePuts.sLine :=strParameterLine;
		fbFilePuts.bExecute:= TRUE;
		Step := 20;
20:
		IF ( NOT fbFilePuts.bBusy ) THEN
			IF ( fbFilePuts.bError ) THEN
				 nErrorID  :=ErrID_9 ;
				bError := TRUE;
				Step := 999;
			ELSE
				Step := 21;
			END_IF
		END_IF

21:	(* Next Line *)
	IF (m+1 <= (nMaxParameters-1) AND m+1 <= nNumParameters) THEN
		m := m+1;
		fbFilePuts.bExecute:= FALSE;
		Step := 19;
	ELSE
		fbFilePuts.bExecute:= FALSE;
		Step := 22;
	END_IF

22:	(* Write footer *)
	fbFilePuts.sLine :='$NEnde';
	fbFilePuts.bExecute:= TRUE;
	Step := 23;

23:
	IF ( NOT fbFilePuts.bBusy ) THEN
		IF ( fbFilePuts.bError ) THEN
			 nErrorID  :=ErrID_9 ;
			bError := TRUE;
			Step := 999;
		ELSE
			fbFileClose.bExecute:=FALSE;
			Step := 30;
		END_IF
	END_IF


30:	(* Close File *)
	fbFileClose.sNetId:='';
	fbFileClose.hFile:=hFileOutput;
	fbFileClose.bExecute:=TRUE;
	fbFileClose.tTimeout:=t#1s;

	IF ( NOT fbFileClose.bBusy ) THEN
		IF ( fbFileClose.bError ) THEN
			 nErrorID  :=ErrID_9 ;
			bError := TRUE;
			Step := 999;
		ELSE
			hFileOutput := 0;
			Step := 35;
		END_IF
	END_IF

	35:
		CASE eParameterType OF
			CNC_AxisParameter:
				Step := 60;
			CNC_ChannelParameter:
				Step := 60;
			CNC_ToolParameter:
				Step := 60;
			CNC_ClampPosition:
				Step := 60;
			CNC_ZeroOffsets:
				Step := 60;
		END_CASE

	40:	(* logical axis ID*)
		TimeOut(IN:=FALSE);
		FbAdsWrite( Port := 553, IdxGrp := nAdsIndexGroup  + nLogChannelID, IdxOffs := (nAdsIndexOffsetlogAxisNumber), LEN := SIZEOF(nLogAxisID), SrcAddr := ADR(nLogAxisID),TMOUT := T#1S, WRITE := TRUE);
		Step := 50;
	50:
		TimeOut(IN:=TRUE, PT:=T#2S);

		FbAdsWrite();
		IF FbAdsWrite.BUSY = FALSE THEN
			IF NOT FbAdsWrite.ERR THEN
				FbAdsWrite( WRITE := FALSE);
				Step := 60;
			ELSE
				FbAdsWrite( WRITE := FALSE);
				nErrorID := ErrID_3;
				Step := 999;
			END_IF
		END_IF

		(* error timeout *)
		IF TimeOut.Q THEN
			nErrorID 	:= ErrID_1;
			Step   	:= 999;
		END_IF

	60:	(* activate List File *)
		TimeOut(IN:=FALSE);

		CASE eParameterType OF

		CNC_AxisParameter:
			FbAdsWrite( Port := nAdsPortNumber, IdxGrp := nAdsIndexGroupAxisParameter  + nLogAxisId, IdxOffs := (nAdsIndexOffsetAxisParameter), LEN := SIZEOF(strFileName), SrcAddr := ADR(strFileName), WRITE := TRUE);
		CNC_ChannelParameter:
			FbAdsWrite( Port := nAdsPortNumber, IdxGrp := nAdsIndexGroup  + nLogChannelID, IdxOffs := (nAdsIndexOffsetChannelParameter), LEN := SIZEOF(strFileName), SrcAddr := ADR(strFileName), WRITE := TRUE);
		CNC_ToolParameter:
			FbAdsWrite( Port := nAdsPortNumber, IdxGrp := nAdsIndexGroup  + nLogChannelID, IdxOffs := (nAdsIndexOffsetToolParameter), LEN := SIZEOF(strFileName), SrcAddr := ADR(strFileName), WRITE := TRUE);
		CNC_ClampPosition:
			FbAdsWrite( Port := nAdsPortNumber, IdxGrp := nAdsIndexGroup  + nLogChannelID, IdxOffs := (nAdsIndexOffsetClampPosition), LEN := SIZEOF(strFileName), SrcAddr := ADR(strFileName), WRITE := TRUE);
		CNC_ZeroOffsets:
			FbAdsWrite( Port := nAdsPortNumber, IdxGrp := nAdsIndexGroup  + nLogChannelID, IdxOffs := (nAdsIndexOffsetZeroOffsets), LEN := SIZEOF(strFileName), SrcAddr := ADR(strFileName), WRITE := TRUE);
		END_CASE

		Step := 70;
	70:
		TimeOut(IN:=TRUE, PT:=T#2S);
		FbAdsWrite();
		IF FbAdsWrite.BUSY = FALSE THEN

			IF NOT FbAdsWrite.ERR THEN
				FbAdsWrite( WRITE := FALSE);
				Step := 0;
			ELSE
				FbAdsWrite( WRITE := FALSE);
				nErrorID := ErrID_4;
				Step := 999;
			END_IF
		END_IF

		(* error timeout *)
		IF TimeOut.Q THEN
			nErrorID 	:= ErrID_1;
			Step   	:= 999;
		END_IF

999: (* Fehler *)
		bBusy  := FALSE;
		bError := TRUE;
		Step 	 := 0;
END_CASE

fbFileOpen();
fbFilePuts();
fbFileClose();

END_FUNCTION_BLOCK

// CNC/11 Util/FB_Uint_Udint
FUNCTION_BLOCK FB_Uint_Udint
VAR
	nOldValue: UINT;
	nDiff: DINT;
	nMinus: BOOL;
	nPlus: BOOL;
END_VAR
VAR_INPUT
	nInSmall: UINT;
END_VAR

VAR_IN_OUT
	nBig: UDINT;
END_VAR

nDiff := nInSmall - nOldValue;


(* Richtung Minus *)
IF ndiff > 10000 THEN
	nBig := nBig - 1;
	nMinus := TRUE;
END_IF

(* Richtung Plus *)
IF ndiff < -10000 THEN
	nBig := nBig + 1;
	nPlus := TRUE;
END_IF

IF (ndiff < 500) AND ndiff > -500 THEN
  nBig := DINT_TO_UDINT( UDINT_TO_DINT(nBig) + nDiff) ;
END_IF
nOldValue := nInSmall;

END_FUNCTION_BLOCK

// CNC/11 Util/HLI3_FindAxisNameAndChannel
FUNCTION HLI3_FindAxisNameAndChannel : BOOL
VAR_INPUT
	LogAxeNr		: UDINT;
	pAxisName		: POINTER TO STRING(HLI_ACHS_NAME_LAENGE);
	pChannelNr		: POINTER TO UINT;
END_VAR
VAR
	i				: UDINT;
	
	pString			: POINTER TO STRING;
END_VAR

FOR i := 0 TO gNrAx - 1 DO
	IF gpAx[i]^.ipo_state.log_achs_nr_r = LogAxeNr THEN
		pChannelNr^ := gpAx[i]^.ipo_state.cnc_channel_r;	(* channel of axis *)
		FOR i := 0 TO INT_TO_UDINT(HLI_CH_AX_MAXIDX) DO
			IF gpCh[pChannelNr^-1]^.bahn_state.coord_r[i].log_achs_nr_r = LogAxeNr THEN
				pString                := ADR(gpCh[pChannelNr^-1]^.bahn_state.coord_r[i].axis_name_r.zeichen);	(* name of axis *)
				pAxisName^             := pString^;
				HLI3_FindAxisNameAndChannel := TRUE;
				RETURN;
			END_IF
		END_FOR
	END_IF
END_FOR

pAxisName^ := '';
pChannelNr^ := 0;
HLI3_FindAxisNameAndChannel := FALSE;

END_FUNCTION

// CNC/11 Util/HLI3_FindHliAxisIdx
FUNCTION HLI3_FindHliAxisIdx : DINT
VAR_INPUT
	nLogAxisNo		: UDINT;	
END_VAR
VAR
	i				: UINT;	
END_VAR

IF nLogAxisNo > MAX_SYS_LOG_AXIS_INDEX OR nLogAxisNo < 1 THEN 
	HLI3_FindHliAxisIdx := -1;
ELSE
	HLI3_FindHliAxisIdx := CNCSystem.LogAxisNo[nLogAxisNo].nHliAxisIdx;	
END_IF

END_FUNCTION

// CNC/11 Util/HLI3_GetEtherCATAxisInfo
FUNCTION HLI3_GetEtherCATAxisInfo : ST_DriveRef
VAR
	arrTemp: ARRAY[1..24] OF BYTE;
	arrNetIdAchse2: ARRAY[0..MAX_STRING_LENGTH] OF BYTE;
	i: INT;
	id: DINT;
	nCha: UINT;
	nPort: UINT;
END_VAR
VAR_INPUT
	nHliAxisIdx: INT;
END_VAR

(* ========================================================= *)
(*    FUN: HLI_GetEtherCATAxisInfo                   		 *)
(* --------------------------------------------------------- *)
(*   Desc: Gets the information about a SoE Drive (Ax5000)   *)
(*  benötigt: TcEtherCAT.lib   *)
(* Return: Structure with the information for the drive     *)
(* Author: MiB                                               *)
(*   Date: 20.11.2012                                        *)
(*   Rev.: 1.2                                               *)
(* ========================================================= *)


IF NOT HLI3_CheckAxisValid(nHliAxisIdx := nHliAxisIdx) THEN
	HLI3_GetEtherCATAxisInfo.sNetId := '';
	HLI3_GetEtherCATAxisInfo.nDriveNo := 0;
	HLI3_GetEtherCATAxisInfo.nSlaveAddr := 0;
	RETURN;	
END_IF


HLI3_GetEtherCATAxisInfo.sNetId := gpAx[nHliAxisIdx]^.lr_state.twincat_box.ads_netid_r;
HLI3_GetEtherCATAxisInfo.nDriveNo := UINT_TO_BYTE(gpAx[nHliAxisIdx]^.lr_state.twincat_box.channel_r);
HLI3_GetEtherCATAxisInfo.nSlaveAddr :=gpAx[nHliAxisIdx]^.lr_state.twincat_box.ads_port_r;

RETURN;

END_FUNCTION

// CNC/11 Util/HLI3_SoftwareLimitSwitches
///*********************************************************************************************************
///NAME.......................:		HLI3_SoftwareLimitSwitches
///DATUM....................:		22.12.2017
///AUTOR....................:		Thomas Voß
///VERSION................:			1.1
///
///Description.: 	Read and Write Software Limit Switches					
///**********************************************************************************************************

FUNCTION_BLOCK HLI3_SoftwareLimitSwitches
VAR_INPUT
	nChannelId		: UINT;
	nLogAxisId		: UINT;	
	fSWLimitNeg		: LREAL;
	fSWLimitPos		: LREAL;
	bExecute		: BOOL;
	/// Windows temp file for sub lists
	strTempPath: STRING;
END_VAR
VAR_OUTPUT
	bBusy  : BOOL;
	bError : BOOL;
	ErrID  :  INT;
END_VAR
VAR
	fbOnTrigger		:  	R_TRIG;

	Step 			: 	UDINT;
		/// Text To File 
	fbFileOpen		: 	FB_FileOpen;
	fbFileRead		: 	FB_FileRead;
	fbFilePuts		: 	FB_FilePuts;
	fbFileClose		: 	FB_FileClose;
	hFileOutput		: 	UINT := 0;
	FbAdsWrite		: 	ADSWRITE;
	FbAdsRead		: 	ADSREAD;
	text			:	STRING(255);
	file			:	STRING(255);
	nSETSWLimitNegValue	: DINT;
	nSETSWLimitPosValue	: DINT;
	Get_SWLimitNeg 	: 	DINT;
	Get_SWLimitPos  : 	DINT;
	offset 			: 	UDINT;
	TimeOut 		: 	TON;	
END_VAR

VAR CONSTANT
	ErrID_1:								INT := 1;		(* Time Out Error *)
	ErrID_2:								INT := 2;		(* Fehler beim Öffnen der Parameterdatei *)
	ErrID_3:								INT := 3;		(* ADS - Fehler : Vorgabe Achs ID *)
	ErrID_4:								INT := 4;		(* ADS - Fehler : Aktivierung der Parameterliste *)
	ErrID_5:								INT := 5;		(* ADS - Fehler :Fehler beim Lesen vom negativen Endschalter  *)
	ErrID_6:								INT := 6;		(* ADS - Fehler :Fehler beim Lesen vom positiven Endschalter  *)
	ErrID_7:								INT := 7;		(* Fehler : Set - SW Limit Switch <> Get SW Limit Switch   *)
	ErrID_9:								INT := 9;		(* File Write Error *)
	ErrID_10:								INT := 10;		(* Invalid AxisId *)
	ErrID_11:								INT := 11;		(* Invalid Limit Parameters *)
	ErrID_12:								INT := 12;		(* No File Path configured*)
	ErrID_13:								INT := 13;		(* Invalid ChannelId *)
END_VAR

fbOnTrigger(CLK:= bExecute);

IF fbOnTrigger.Q THEN
	Step 	:= 10;
	ErrID 	:= 0;
	bError	 := 0;
	bBusy := TRUE;
END_IF

CASE Step OF
0:
	bBusy := FALSE;

10:		// Check Input Parameters 
		nSetSWLimitNegValue	:= LREAL_TO_DINT(fSWLimitNeg*10000);
		nSetSWLimitPosValue	:= LREAL_TO_DINT(fSWLimitPos*10000);
		
		IF (nLogAxisId < 0) THEN
			bError :=	TRUE;
			ErrID  :=  ErrID_10;
			Step   := 999;
		ELSIF  (nLogAxisId > MAX_SYS_LOG_AXIS_INDEX) THEN
			bError :=	TRUE;
			ErrID  :=  ErrID_10;
			Step   := 999;
		ELSIF (CNCSystem.LogAxisNo[nLogAxisId].nHliAxisIdx = -1) THEN
			bError :=	TRUE;
			ErrID  :=  ErrID_10;
			Step   := 999;
		ELSIF (nSETSWLimitNegValue > nSetSWLimitPosValue) OR (nSETSWLimitNegValue = nSetSWLimitPosValue) THEN	
			bError :=	TRUE;
			ErrID  :=   ErrID_11;
			Step   :=   999;
		ELSIF (strTempPath = '') THEN
			bError :=	TRUE;
			ErrID  :=   ErrID_12;
			Step   :=   999;
		ELSIF (nChannelId < 1 OR UINT_TO_INT(nChannelId) > HLI_SYS_CH_MAXIDX+1) THEN
			bError :=	TRUE;
			ErrID  :=   ErrID_13;
			Step   :=   999; 
		ELSE
			Step 	:= 20;		
		END_IF		
					
20:
		file := CONCAT(strTempPath, '\axis');
		file := CONCAT(file, UINT_TO_STRING(nLogAxisId));
		file := CONCAT(file, '.lis');
								
		text := 'kopf.achs_nr ';
		text := CONCAT(text, UINT_TO_STRING(nLogAxisId));
		text := CONCAT(text, '$Nkenngr.swe_neg    ');
		text := CONCAT(text, DINT_TO_STRING(nSetSWLimitNegValue));
		text := CONCAT(text, '$Nkenngr.swe_pos    ');
		text := CONCAT(text, DINT_TO_STRING(nSetSWLimitPosValue));
		text := CONCAT(text, '$NEnde');

		TimeOut(IN:=FALSE);
		fbFileOpen.bExecute := FALSE;
		Step := Step+10;
					
30:	(* write file to destination folder *)
	fbFileOpen.sNetId := '';
	fbFileOpen.sPathName := file;
	fbFileOpen.nMode := FOPEN_MODEWRITE OR FOPEN_MODETEXT;
	fbFileOpen.ePath := PATH_GENERIC;
	fbFileOpen.tTimeout := t#1s;
	fbFileOpen.bExecute := TRUE;
	Step := Step+10;

40:
	IF ( NOT fbFileOpen.bBusy ) THEN
		IF ( fbFileOpen.bError ) THEN
			ErrID  :=ErrID_9 ;
			bError := TRUE;
			Step := 999;
		ELSE
			hFileOutput := fbFileOpen.hFile;
			fbFilePuts.bExecute:= FALSE;
			Step := Step+10;
		END_IF
	END_IF

50: (* Write Header File *)
	fbFilePuts.sNetId:='';
	fbFilePuts.hFile:=hFileOutput;
	fbFilePuts.bExecute:=TRUE;
	fbFilePuts.tTimeout:=t#10s;
	fbFilePuts.sLine :=text;
	Step := Step+10;

60:
	IF ( NOT fbFilePuts.bBusy ) THEN
		IF ( fbFilePuts.bError ) THEN
			ErrID  :=ErrID_9 ;
			bError := TRUE;
			Step := 999;
		ELSE
			fbFilePuts.bExecute:= FALSE;		
			Step := Step+10;
		END_IF
	END_IF

70:
	IF ( NOT fbFilePuts.bBusy ) THEN
		IF ( fbFilePuts.bError ) THEN
			ErrID  :=ErrID_9 ;
			bError := TRUE;
			Step := 999;
		ELSE
			fbFileClose.bExecute:=FALSE;
			Step := Step+10;
		END_IF
	END_IF


80:	(* Close File *)
	fbFileClose.sNetId:='';
	fbFileClose.hFile:=hFileOutput;
	fbFileClose.bExecute:=TRUE;
	fbFileClose.tTimeout:=t#1s;

	IF ( NOT fbFileClose.bBusy ) THEN
		IF ( fbFileClose.bError ) THEN
			ErrID  :=ErrID_9 ;
			bError := TRUE;
			Step := 999;
		ELSE
			hFileOutput := 0;
			Step := Step+10;
		END_IF
	END_IF
		
90:		(* logical axis ID*)
		TimeOut(IN:=FALSE);
		FbAdsWrite( Port := 553, IdxGrp := 16#20100 + nChannelId, IdxOffs := (16#37), LEN := SIZEOF(nLogAxisId), SrcAddr := ADR(nLogAxisId),TMOUT := T#1S, WRITE := TRUE);
		Step := Step+10;
100:
		TimeOut(IN:=TRUE, PT:=T#2S);

		FbAdsWrite();
		IF FbAdsWrite.BUSY = FALSE THEN
			IF NOT FbAdsWrite.ERR THEN
				FbAdsWrite( WRITE := FALSE);
				Step := Step+10;
			ELSE
				FbAdsWrite( WRITE := FALSE);
				ErrID := ErrID_3;
				Step := 999;
			END_IF
		END_IF

		(* error timeout *)
		IF TimeOut.Q THEN
			ErrID 	:= ErrID_1;
			Step   	:= 999;
		END_IF

110:		(* Achsparameter aktivieren *)
		TimeOut(IN:=FALSE);

	    FbAdsWrite( WRITE := FALSE);
		FbAdsWrite( Port := 553, IdxGrp := 16#20100 + nChannelId, IdxOffs := (16#36), LEN := SIZEOF(file), SrcAddr := ADR(file), WRITE := TRUE);
		Step := Step+10;
		
120:
		TimeOut(IN:=TRUE, PT:=T#2S);
		FbAdsWrite();
		IF FbAdsWrite.BUSY = FALSE THEN

			IF NOT FbAdsWrite.ERR THEN
				FbAdsWrite( WRITE := FALSE);
				FbAdsRead(Read:=FALSE);
				Step := Step+10;
			ELSE
				FbAdsWrite( WRITE := FALSE);
				ErrID := ErrID_4;
				Step := 999;
			END_IF
		END_IF

		(* error timeout *)
		IF TimeOut.Q THEN
			ErrID 	:= ErrID_1;
			Step   	:= 999;
		END_IF

130: (* Read negative Limit Switch *)
	TimeOut(IN:=FALSE);
	FbAdsRead(	NETID:= '',				(* local *)
				PORT:= 553,					(* Port number of Task COM, all ADS-Requests to the NC-kernel  *)										(* must sent to this port                                      *)
				IDXGRP:=16#00020200+nLogAxisId,    (*  *)
				IDXOFFS:= 16#26,
				LEN:=SIZEOF(Get_SWLimitNeg),		(* number of bytes that shall be read                          *)
				DESTADDR:= ADR(Get_SWLimitNeg),  (* memory for the read value, must be provided by the user     *)
				READ:=TRUE,					(* a rising edge on this input starts the read request         *)
				TMOUT:= T#1s);       (* maximum time for read request                               *)

		Step := Step+10;

140:
		TimeOut(IN:=TRUE, PT:=T#2S);
		FbAdsRead();
		IF NOT FbAdsRead.Busy THEN
			IF NOT FbAdsRead.ERR THEN
				FbAdsRead(READ := FALSE);
				Step := Step+10;
			ELSE
				FbAdsRead(READ := FALSE);
				ErrID 	:= ErrID_5;
				Step := 999;
			END_IF
		END_IF

		(* error timeout *)
		IF TimeOut.Q THEN
			ErrID 	:= ErrID_1;
			Step   	:= 999;
		END_IF



150: (* Read positive Limit Switch *)
	TimeOut(IN:=FALSE);
	FbAdsRead(	NETID:= '',				(* local *)
				PORT:= 553,					(* Port number of Task COM, all ADS-Requests to the NC-kernel  *)										(* must sent to this port                                      *)
				IDXGRP:=16#00020200+nLogAxisId,    (*  *)
				IDXOFFS:= 16#25,
				LEN:=SIZEOF(Get_SWLimitPos),		(* number of bytes that shall be read                          *)
				DESTADDR:= ADR(Get_SWLimitPos),  (* memory for the read value, must be provided by the user     *)
				READ:=TRUE,					(* a rising edge on this input starts the read request         *)
				TMOUT:= T#1s);       (* maximum time for read request                               *)
	Step := Step+10;

160:	TimeOut(IN:=TRUE, PT:=T#2S);
		FbAdsRead();
		IF NOT FbAdsRead.Busy THEN
			IF NOT FbAdsRead.ERR THEN
				FbAdsRead(READ := FALSE);
				Step := Step+10;
			ELSE
				FbAdsRead(READ := FALSE);
				ErrID 	:= ErrID_6;
				Step := 999;
			END_IF
		END_IF

170:	(* Check *)
		IF (Get_SWLimitNeg = nSetSWLimitNegValue) AND (Get_SWLimitPos = nSetSWLimitPosValue) THEN
			bBusy := FALSE;
			Step := 0;
		ELSE
			ErrID 	:= ErrID_7;
			Step := 999;
		END_IF


999: (* Fehler *)
		bBusy  := FALSE;
		bError := TRUE;
		Step 	 := 0;
END_CASE

fbFileOpen();
fbFilePuts();
fbFileClose();

END_FUNCTION_BLOCK

// CNC/12 CNC_Axis/FB_ActivateCompTable
(**********************************************************************************************************
NAME...................:		FB_ActivateSSFK	
DATUM..................:		23.01.2009
AUTOR..................:		Thomas Voß
VERSION................:		1.0

BESCHREIBUNG.:	Aktiviert Korrekturwerttabelle über den CNC List File Interpreter
......................: 	

***********************************************************************************************************)
FUNCTION_BLOCK FB_ActivateCompTable
VAR_INPUT
	bExecute			: BOOL;
	strPathCompTable 	: STRING(256);
	nAxisID				: DINT;
	tTimeout			: TIME := T#10S;
END_VAR
VAR_OUTPUT
	bBusy			: 	BOOL;
	bError			:	BOOL;
	nErrID			:	UDINT;
END_VAR
VAR
	iState 			:  UINT;
	fbOnTrigger		:  R_TRIG;
	fbAdsWrite		:  ADSWRITE;
END_VAR

fbOnTrigger(CLK:= bExecute);

CASE iState OF

0 :

	bBusy := FALSE;

	IF fbOnTrigger.Q THEN
			iState := 10;
			nErrID := 0;
			bError := 0;
			bBusy := TRUE;
			fbAdsWrite(WRITE := FALSE);
		END_IF


10:                (* logical axis ID*)
                fbAdsWrite( Port := 553, IdxGrp := 16#20101, IdxOffs := (16#3A), LEN := SIZEOF(nAxisID), SrcAddr := ADR(nAxisID), WRITE := TRUE);

		IF NOT fbAdsWrite.Busy THEN
			IF fbAdsWrite.Err THEN
				bError := fbAdsWrite.Err;
				nErrID :=fbAdsWrite.ERRID;
				iState := 0;
			ELSE
				fbAdsWrite(WRITE := FALSE);
				iState := 20;
			END_IF
		END_IF


20: (* Korrekturwert Tabelle aktivieren *)

                FbAdsWrite( Port := 553, IdxGrp := 16#20101, IdxOffs := (16#39), LEN := SIZEOF(strPathCompTable), SrcAddr := ADR(strPathCompTable), WRITE := TRUE);

		IF NOT fbAdsWrite.Busy THEN
			IF fbAdsWrite.Err THEN
				bError := fbAdsWrite.Err;
				nErrID :=fbAdsWrite.ERRID;
				iState := 0;
			ELSE
				fbAdsWrite(WRITE := FALSE);
				iState := 0;
			END_IF
		END_IF

END_CASE

END_FUNCTION_BLOCK

// CNC/12 CNC_Axis/FB_CNCAxis
FUNCTION_BLOCK FB_CNCAxis EXTENDS HLI3_CNCAxisBase
VAR_INPUT
	nLogAxisNo : INT;
END_VAR
VAR_OUTPUT
END_VAR
VAR
END_VAR

(* ========================================================= *)
(*     FB: FB_CNCAxis                                  		 *)
(* --------------------------------------------------------- *)
(*   Desc:  CNC Axis Control							   	 *)
(*   Author: TV				                                 *)
(*   Date: 2018.01.25                                        *)
(*   Rev.: 1.0                                               *)
(* ==========================================================*)

IF nLogAxisNo < 1 OR  nLogAxisNo > UINT_TO_INT(MAX_SYS_LOG_AXIS_INDEX) THEN
	RETURN;
END_IF

IF CNCSystem.LogAxisNo[nLogAxisNo].nHliAxisIdx = -1 THEN
	RETURN;
END_IF

SUPER^(nHliIdx := CNCSystem.LogAxisNo[nLogAxisNo].nHliAxisIdx);

END_FUNCTION_BLOCK

// CNC/12 CNC_Axis/HLI3_CNCAxisBase
FUNCTION_BLOCK HLI3_CNCAxisBase
VAR_INPUT
	{attribute 'hide'}
	nHliIdx						: INT;
	bEnable 					: BOOL;	
  //  bEnablePositive 			: BOOL; 
  //  bEnableNegative 			: BOOL; 
	bCalibrationCam				: BOOL;		
	bSetRefOffset				: BOOL;
	fRefOffset					: LREAL;  // [ mm or degree ]
	bFeedhold				 	: BOOL;
	stOptions           		: ST_CNC_AX_Options;	
	stParameter					: ST_CNC_AX_Parameter;
	stPLCopen					: ST_CNC_AX_PLCopen;
END_VAR
VAR_OUTPUT
	stStatus					: ST_CNC_AX_Status;	
END_VAR
VAR
	fbSetAxisRelease 			: HLI3_SetAxisRelease;
	fbSetAxisReferenceOffset	: HLI3_SetAxisReferenceOffset;
	fbActivateCompTable			: FB_ActivateCompTable;
	bInit 						: BOOL;
	fbOnTrigger					: R_TRIG;
	nStepWriteParam				: INT;
	fbOnTriggerCompTable		: R_TRIG;
	nStepActivateCompTable      : INT;
	
	// PLCopen Platform
	fbMC_SetOverride			: MC_SetOverride;
	fbMC_Home					: MC_Home;
	fbMC_MoveAbsolute			: MC_MoveAbsolute;
	fbMC_ReadAxisError 			: MC_ReadAxisError;	
	fbMC_Stop					: MC_Stop;
	fbMC_Reset					: MC_Reset;		
END_VAR

(* ========================================================= *)
(*     FB: FB_CNCAxis                                  		 *)
(* --------------------------------------------------------- *)
(*   Desc:  CNC Axis Control							   	 *)
(*   Author: TV				                                 *)
(*   Date: 2018.03.19                                        *)
(*   Rev.: 1.4                                               *)
(* ==========================================================*)

IF NOT CNCSystem.bHLIInit THEN
	RETURN;
END_IF

IF NOT (HLI3_CheckAxisValid(nHliAxisIdx := nHliIdx)) THEN
	RETURN;
END_IF

ACT_Init();
ACT_Parameter();
ACT_Status();
ACT_Options();
ACT_PLCopen();

// Axis Release
fbSetAxisRelease(
	bEnable:= bEnable, 
	nHliAxisIdx:= nHliIdx, 
	bAxisHasError => stStatus.bHasError,
	bAxisIsEnabled => stStatus.bIsEnabled,
	bAxisIsReady => stStatus.bIsReady
);
	
// Reference Cam        
HLI3_SetAxisReferenceCam(nHliIdx,bCalibrationCam);

// Set Ref. Offset
fbSetAxisReferenceOffset(
	Execute:= bSetRefOffset, 
	nHliAxisIdx:= nHliIdx, 
	nOffset:= fRefOffset);

// Axis Feedhold	
HLI3_SetAxisFeedhold(nHliIdx,bFeedhold);

ACTION ACT_Init:
IF NOT bInit THEN
	gpAX[nHliIdx]^.ipo_mc_control.reduced_speed.enable_w := TRUE;
	gpAX[nHliIdx]^.ipo_mc_control.reduced_speed_zone.enable_w := TRUE;
	gpAX[nHliIdx]^.ipo_mc_control.reduced_speed_2_zone.enable_w := TRUE;
END_IF
END_ACTION

ACTION ACT_Options:
// Clear Reference Position
HLI3_ClearReferencePosition(nHliAxisIdx := nHliIdx, bExecute := stOptions.bResetCalibration);

// Probing Signal       
HLI3_SetProbingSignal(nHliIdx,stOptions.bProbingSignal);

// Reduced_Speed
gpAX[nHliIdx]^.ipo_mc_control.reduced_speed.command_w := stOptions.bReducedSpeed;

// Reduced_Speed Zone 1
gpAX[nHliIdx]^.ipo_mc_control.reduced_speed_zone.command_w := stOptions.bReducedSpeedZone1;

// Reduced_Speed Zone 2
gpAX[nHliIdx]^.ipo_mc_control.reduced_speed_2_zone.command_w := stOptions.bReducedSpeedZone2;
 
// Activate Compensation Table
fbOnTriggerCompTable(CLK:= stOptions.bActivateCompTable);

IF fbOnTriggerCompTable.Q THEN
	nStepActivateCompTable:= 10;
END_IF

CASE nStepActivateCompTable OF
0:
	;
10:
	IF NOT fbActivateCompTable.bBusy AND NOT bCNC_AX_ActivateCompTableLock  THEN
			bCNC_AX_ActivateCompTableLock  := TRUE;						 
			fbActivateCompTable.bExecute:= FALSE;	 
			nStepActivateCompTable := 20;	
	END_IF	
20:			
	fbActivateCompTable.bExecute:= TRUE;
    fbActivateCompTable.strPathCompTable:= stOptions.strPathCompTable; 
	fbActivateCompTable.nAxisID:= gpAx[nHliIdx]^.head.log_ax_nr_r;	
	nStepActivateCompTable := 30;			 				
	
30:	IF NOT fbActivateCompTable.bBusy OR  fbActivateCompTable.bError THEN		
		bCNC_AX_ActivateCompTableLock := FALSE;
		nStepActivateCompTable := 0;		
	END_IF
	
END_CASE
END_ACTION

ACTION ACT_Parameter:


fbOnTrigger(CLK:= stParameter.bWriteParameter);

IF fbOnTrigger.Q THEN
	nStepWriteParam := 10;
END_IF

CASE nStepWriteParam OF
0:
	;
10:
	IF NOT fbCNC_AX_WriteParameter.bBusy AND NOT bCNC_AX_WriteParameterLock THEN
			bCNC_AX_WriteParameterLock := TRUE;						 
			fbCNC_AX_WriteParameter.bExecute:= FALSE;	 
			nStepWriteParam := 20;	
	END_IF
	
20:			 
			fbCNC_AX_WriteParameter.nLogChannelID:= 1;		 
			fbCNC_AX_WriteParameter.nLogAxisId:= gpAx[nHliIdx]^.head.log_ax_nr_r; 
			fbCNC_AX_WriteParameter.bExecute:= TRUE; 
			fbCNC_AX_WriteParameter.nNumParameters:= stParameter.nNumParameters;
			fbCNC_AX_WriteParameter.eParameterType:= E_CNCParameterTypes.CNC_AxisParameter; 
			fbCNC_AX_WriteParameter.strTempPath:= stParameter.strTempPath; 		 
			fbCNC_AX_WriteParameter.stParameter:= stParameter.ParamList;
			nStepWriteParam := 30;	
	
30:	IF NOT fbCNC_AX_WriteParameter.bBusy OR  fbCNC_AX_WriteParameter.bError THEN		
		bCNC_AX_WriteParameterLock:= FALSE;
		nStepWriteParam := 0;		
	END_IF
	
END_CASE
END_ACTION

ACTION ACT_PLCopen:
IF 	CNCSystem.bPLCopenPlatformInit AND 
	gpAx[nHliIdx]^.lr_state.is_sai_r AND
	g_array_axis_ref[nHliIdx].axsd_state <> MCV_AXSD_STATES.INIT_STATE 	
THEN

(* Override *)
IF stPLCopen.nOverride > 1000 THEN stPLCopen.nOverride := 1000; END_IF  
IF stPLCopen.nOverride < 0 THEN stPLCopen.nOverride := 0; END_IF

fbMC_SetOverride(
	Axis:= g_array_axis_ref[nHliIdx],  
	Enable:= TRUE, 
	VelFactor:= UINT_TO_LREAL(stPLCopen.nOverride) / 1000.0, 
	VelFactorMaxShift:= , 
	Enabled=> , 
	Error=> , 
	ErrorID=> );
	
fbMC_Home(
	Axis:= g_array_axis_ref[nHliIdx], 
	Execute:= stPLCopen.bExecuteHoming, 
	CamSignal:= stPLCopen.bCamSignal,
	Done=> stStatus.PLCopen.bHomingDone,
	CommandAborted=> , 
	Error=> , 
	ErrorID=> );	
	
fbMC_MoveAbsolute(
	Axis:= g_array_axis_ref[nHliIdx], 
	Execute:=  stPLCopen.bExecuteMoveAbsolute, 
	Position:= stPLCopen.fPosition * 10000.0, 
	Velocity:= stPLCopen.fVelocity * 16.6666,
	Acceleration:= stPLCopen.fAcceleration, 
	Deceleration:= stPLCopen.fAcceleration,
	Jerk:= stPLCopen.fJerk, 
	Direction:= stPLCopen.nDirection, 
	Done=> stStatus.PLCopen.bMoveAbsoluteDone, 
	CommandAborted=> , 
	Error=> , 
	ErrorID=> );	
	
	
	fbMC_Stop(
	Axis:= g_array_axis_ref[nHliIdx],  
	Execute:= stPLCopen.bExecuteStop, 
	Deceleration:= stPLCopen.fAcceleration,  
	Jerk:= stPLCopen.fJerk,  
	Done=> stStatus.PLCopen.bStopDone, 
	Error=> , 
	ErrorID=> );
	
	fbMC_Reset(
	Axis:= g_array_axis_ref[nHliIdx], 
	Execute:= stPLCopen.bExecuteReset,  
	Done=> stStatus.PLCopen.bResetDone, 
	Error=> , 
	ErrorID=> );
				
	stStatus.PLCopen.bError := fbMC_SetOverride.Error OR fbMC_MoveAbsolute.Error OR fbMC_Home.Error OR fbMC_Stop.Error OR fbMC_Reset.Error;;

	IF fbMC_SetOverride.ErrorID <> 0 THEN 
		stStatus.PLCopen.nErrorID := fbMC_SetOverride.ErrorID;
	ELSIF fbMC_Reset.ErrorID <> 0 THEN 
		stStatus.PLCopen.nErrorID := fbMC_Reset.ErrorID;
	ELSIF fbMC_Stop.ErrorID <> 0 THEN
		stStatus.PLCopen.nErrorID := fbMC_Stop.ErrorID;
	ELSIF fbMC_Home.ErrorID <> 0 THEN 
		stStatus.PLCopen.nErrorID := fbMC_Home.ErrorID;
	ELSIF fbMC_MoveAbsolute.ErrorID <> 0 THEN  
		stStatus.PLCopen.nErrorID := fbMC_MoveAbsolute.ErrorID;		
	ELSE 		
		stStatus.PLCopen.nErrorID := 0;
	END_IF
	
	IF stStatus.PLCopen.nErrorID = 40001 THEN 
	
		fbMC_ReadAxisError(
			Axis:= g_array_axis_ref[nHliIdx],  
			Enable:= TRUE);
			
			IF fbMC_ReadAxisError.AxisErrorID <> 0 THEN
				stStatus.PLCopen.nErrorID := UDINT_TO_DINT(fbMC_ReadAxisError.AxisErrorID);
			END_IF
			
	END_IF
			
END_IF
END_ACTION

ACTION ACT_Status:
stStatus.bHomingDone := gpAx[nHliIdx]^.lr_state.homing_done_r;

stStatus.fSetPosACS	:= DINT_TO_LREAL(gpAx[nHliIdx]^.lr_state.active_position_acs_r) / 10000.0;;
stStatus.fActPosACS	:= DINT_TO_LREAL(gpAx[nHliIdx]^.lr_state.current_position_acs_r) / 10000.0;


IF (gpAx[nHliIdx]^.ipo_state.spindle_axis_r) THEN // Spindle
	stStatus.fActVelo := DINT_TO_LREAL( gpAx[nHliIdx]^.lr_state.current_rev_r) / 16.66666666 / 360.00;
ELSE
	stStatus.fActVelo := DINT_TO_LREAL( gpAx[nHliIdx]^.lr_state.current_rev_r) / 16.66666666;
END_IF

// CNC Axis Error ID
IF (gpAx[nHliIdx]^.ipo_state.cnc_channel_r > 0 ) THEN

	IF CNCSystem.LogChannelNo[gpAx[nHliIdx]^.ipo_state.cnc_channel_r].nHliChannelIdx <> -1 THEN

		IF gpCh[CNCSystem.LogChannelNo[gpAx[nHliIdx]^.ipo_state.cnc_channel_r].nHliChannelIdx]^.channel_mc_control.mode_and_state.state_r.state = HLI_IMCM_PROCESS_RESETTING THEN
			stStatus.nCNCErrorID := 0;
			CNCSystem.LogAxisNo[gpAx[nHliIdx]^.head.log_ax_nr_r].nCNCErrorID := 0;
		ELSE
			stStatus.nCNCErrorID := CNCSystem.LogAxisNo[gpAx[nHliIdx]^.head.log_ax_nr_r].nCNCErrorID;	
		END_IF

	END_IF
END_IF
END_ACTION

END_FUNCTION_BLOCK

// CNC/3 Control/HLI3_SetAxisReferenceCam
FUNCTION HLI3_SetAxisReferenceCam : BOOL
VAR_INPUT
	nHliAxisIdx: INT;
	bReferenceCam: BOOL;
END_VAR
VAR
	/// Index of axis specific HLI area 
	nHliAxIfcIdx: INT;
END_VAR

(* ========================================================= *)
(*    FUN: HLI_SetAxisReferenceCam                           *)
(* --------------------------------------------------------- *)
(*   Desc:                                                   *)
(* Author: MK,MiB                                            *)
(*   Date: 30.11.2012                                        *)
(*   Rev.: 1.1                                               *)
(* ========================================================= *)


IF NOT HLI3_CheckAxisValid(nHliAxisIdx := nHliAxisIdx) THEN
	HLI3_SetAxisReferenceCam := FALSE;
	RETURN;
END_IF

(* set reference cam *)
gpAx[nHliAxisIdx]^.lr_mc_control.reference_cam.enable_w  := TRUE;
gpAx[nHliAxisIdx]^.lr_mc_control.reference_cam.command_w := bReferenceCam;

HLI3_SetAxisReferenceCam := TRUE;

END_FUNCTION

// CNC/3 Control/HLI3_SetAxisFeedhold
FUNCTION HLI3_SetAxisFeedhold : BOOL
VAR_INPUT
	/// number of Axis 
	nHliAxisIdx: INT;
	bFeedHold: BOOL;
END_VAR

(* ========================================================= *)
(*    FUN: HLI_SetAxisFeedhold                               *)
(* --------------------------------------------------------- *)
(*   Desc: Set the Axis Feedhold                             *)
(* 	 Author: TV                                              *)
(*   Date: 09.05.2018                                        *)
(*   Rev.: 1.0                                               *)
(*   Rev.: 1.1                             					 *)
(* ========================================================= *)
IF NOT (HLI3_CheckAxisValid(nHliAxisIdx := nHliAxisIdx)) THEN
	HLI3_SetAxisFeedhold := FALSE;
	RETURN;
END_IF

gpAx[nHliAxisIdx]^.ipo_mc_control.feedhold.enable_w  := TRUE;
gpAx[nHliAxisIdx]^.ipo_mc_control.feedhold.command_w := bFeedhold;

HLI3_SetAxisFeedhold := TRUE;

END_FUNCTION

// CNC/3 Control/HLI3_SetAxisRelease
FUNCTION_BLOCK HLI3_SetAxisRelease
VAR_INPUT
	bEnable: BOOL;
	nHliAxisIdx: INT;
END_VAR
VAR_OUTPUT
	bAxisIsReady: BOOL;
	bAxisIsEnabled: BOOL;
	bAxisHasError: BOOL;
	nDriveType: UDINT;
	bError: BOOL;
	nErrorId: UDINT;
	nErrorState: UINT;
END_VAR
VAR
	bReadyForPowerOn: BOOL;
	bReadyForControlLoopOn: BOOL;
	nHliAxisIdxOld: INT;
	nState: UINT;
	nStateOld: UINT;
	tActiveTimeOut: TIME := TIME#5s0ms;
	wDriveState: WORD;
	fbTonTimeOut: TON;
END_VAR
VAR CONSTANT
	ERR_INVALID_AXIS_IDX: UDINT := 10000;
	ERR_UNSUPPORTED_DRIVE: UDINT := 10001;
	ERR_TIME_OUT: UDINT := 10002;
END_VAR

(****************************************************************************************)
(* POU:		HLI3_SetAxisRelease                      									*)
(* Type:	Function block																*)
(* Author: 	HR																			*)
(* Date: 	14/01/10																	*)
(* Rev.: 	1.0																			*)
(* ------------------------------------------------------------------------------------ *)
(* Author: 	TV																			*)
(* Date: 	14/04/11																	*)
(* Rev.: 	1.1																			*)
(* 			Implementation for terminal drives											*)
(* ------------------------------------------------------------------------------------ *)
(* Author: 	HR																			*)
(* Date: 	14/08/27																	*)
(* Rev.: 	1.2																			*)
(* 			Fixed terminal drive issue --> According to the ISG docs terminal drives	*)
(*			are supported by means of the torque permission control unit only! There-	*)
(*			fore this has to be switched by the 'bEnable' input. Tested with EL7041		*)
(* ------------------------------------------------------------------------------------ *)
(* Author: 	MiB																			*)
(* Date: 	16/04/06																	*)
(* Rev.: 	1.2																			*)
(* 			Enable follow up only for non simulation axis								*)
(* ------------------------------------------------------------------------------------ *)
(* Author: 	TV																			*)
(* Date: 	18/07/12																	*)
(* Rev.: 	1.4																			*)
(* 			Implementation for ProfiDrives												*)
(* ------------------------------------------------------------------------------------ *)		
(* Desc:	Sets axes release and follow up mode using the axis specific control units 	*)
(*			'.lr_mc_control.torque_permission', 'lr_mc_control.release_feedhold',		*)
(*			'lr_mc_control.drive_on' and 'lr_mc_control.follow_up' depending on the 	*)
(*			subsequent drive type (e.g. Sercos,...). The following drive type are 		*)
(*			supported:																	*)
(*				+ Sercos and SoE														*)
(*				+ CanOpen and CoE (according to CiA402 drive profile)					*)
(*				+ Simulation drives														*)
(*																						*)
(*			This function block may raise the following error numbers					*)
(*				+ 10000	--> Invalid 'nHliAxisIdx'										*)
(*				+ 10001 --> Unsupported drive type										*)
(*				+ 10002 --> Time out while setting axis release							*)
(*																						*)
(*			IMPORTANT: This function block does not implement any state specific en- or	*)
(*			disabling of the drive. It simply tries to enable the subsequent axis as	*)
(*			long as input variable 'bEnable' is TRUE. That means it won´t disable the 	*)
(*			drive in case of any errors or loss prerequisited operation conditions (e.g.*)
(*			power supply). It is assumed that the drive will handle those situations	*)
(*			internally!																	*)
(*				  																		*)
(* 			Tested with following drives:												*)
(*																						*)
(*			VENDOR				MAKE					FW-VERSION			COM-SYS 	*)
(* 			------				----					----------			-------		*)
(* 			Beckhoff			AX5xxx					2.03 (B26)			SoE			*)
(* 			Beckhoff			EL7201					03					CoE			*)
(*			Beckhoff			EL7041					10					Terminal	*)	
(* 			ELMO				Gold					01.01.07.12			CoE			*)
(****************************************************************************************)

(****************************************************************************************)
(*									Check axis index									*)
(****************************************************************************************)
IF NOT HLI3_CheckAxisValid(nHliAxisIdx) THEN
	bError		:= TRUE;
	nErrorId	:= ERR_INVALID_AXIS_IDX;
	RETURN;
END_IF

(****************************************************************************************)
(*										Clear errors									*)
(****************************************************************************************)
IF bError THEN
	CASE nErrorId OF
	 (* -------------------------------------------------------------------------------	*)
	 ERR_INVALID_AXIS_IDX:
	 	(* Reset invalid HLI axis index error as soon as this line has been hit!		*)
		AC_ClearError();
		
	(* -------------------------------------------------------------------------------	*)
	 ERR_UNSUPPORTED_DRIVE:
		(* Reset unsupported drive type error in case the HLI axis index has been 		*)
		(* changed!																		*)
		IF (nHliAxisIdx <> nHliAxisIdxOld) THEN
			nHliAxisIdxOld	:= nHliAxisIdx;
			AC_ClearError();
		END_IF
 
	(* -------------------------------------------------------------------------------	*) 
	 ERR_TIME_OUT:
 		(* Will be resetted individually by each drive type specific action!			*)
	END_CASE
END_IF

(****************************************************************************************)
(*								Switch follow up mode 									*)
(****************************************************************************************)
IF gpAx[nHliAxisIdx]^.lr_state.drive_type_r = 4 THEN   (* type == 4 -> simulation axis -> don't enable follow up mode *)
	gpAx[nHliAxisIdx]^.lr_mc_control.follow_up.command_w := FALSE;
ELSE
	gpAx[nHliAxisIdx]^.lr_mc_control.follow_up.command_w := NOT bEnable;
END_IF

(****************************************************************************************)
(*						Copy axis state information to local variables					*)
(****************************************************************************************)
wDriveState				:= gpAx[nHliAxisIdx]^.lr_state.native_drive_state_r;
nDriveType				:= gpAx[nHliAxisIdx]^.lr_state.drive_type_r;
bAxisHasError			:= gpAx[nHliAxisIdx]^.lr_state.error_r;
bReadyForPowerOn		:= gpAx[nHliAxisIdx]^.lr_state.ready_for_power_on_r;
bReadyForControlLoopOn	:= gpAx[nHliAxisIdx]^.lr_state.ready_for_control_loop_on_r;

(****************************************************************************************)
(*							 Constant timeout implementation							*)
(****************************************************************************************)
IF (nStateOld <> nState) THEN
	nStateOld	:= nState;
	fbTonTimeOut(IN := FALSE);
END_IF

fbTonTimeOut
	(IN := TRUE,
	 PT := tActiveTimeOut
	);

(****************************************************************************************)
(*								Drive type specific axis release						*)
(****************************************************************************************)
CASE nDriveType OF
	HLI_DRIVE_CANOPEN	: AC_CanOpenDrive();
	HLI_DRIVE_SERCOS	: AC_SercosDrive();
	HLI_DRIVE_SIMU		: AC_SercosDrive();
	HLI_DRIVE_TERMINAL  : AC_TerminalDrive();
	HLI_DRIVE_PROFIDRIVE: AC_ProfiDrive();
ELSE
	bError				:= TRUE;
	nErrorId			:= ERR_UNSUPPORTED_DRIVE;
END_CASE

ACTION AC_CanOpenDrive:
(****************************************************************************************)
(*										Status data										*)
(****************************************************************************************)
(* Ready state is signalled if the drive´s state is unequal to 'Not ready to switch on'	*)
bAxisIsReady	:= bReadyForControlLoopOn; 
 
(* Enabled state is derived from state 'Operation enabled' (information provided via	*)
(* HLI) and from status word bit no. 01 (switched on)!									*)
bAxisIsEnabled	:= bReadyForControlLoopOn AND bReadyForPowerOn AND wDriveState.1;

(****************************************************************************************)
(*						Command data (CanOpen requires a state machine)					*)
(****************************************************************************************)
(* Switch back to initial state in case the user want´s to disable the drive or an axis	*)
(* error occured, which requires a new srun of the sequence!							*)
IF NOT bEnable OR wDriveState.3 THEN
	nState				:= 0;
END_IF

CASE nState OF
 (* -----------------------------------------------------------------------------------	*)
 0: (* INIT *)
 	gpAx[nHliAxisIdx]^.lr_mc_control.torque_permission.command_w	:= FALSE;
 	gpAx[nHliAxisIdx]^.lr_mc_control.release_feedhold.command_w		:= FALSE;
	
	(* Start sequence in case the user wants to enable the drive and there is no error.	*)
 	IF bEnable AND NOT wDriveState.3 AND bAxisIsReady THEN
		(* Set time out once! *)
		tActiveTimeOut	:= T#2S;	
	
		// Switch on disabled???
		IF wDriveState.6 THEN
			nState		:= 10;
		//Ready to switch on???
		ELSIF wDriveState.0 THEN
			nState		:= 20;
		//Switched on???
		ELSIF wDriveState.1 THEN
			nState		:= 30;
		//Operation enabled???
		ELSIF wDriveState.2 THEN
			nState		:= 40;
		END_IF
	END_IF
	
 (* -----------------------------------------------------------------------------------	*)
 10: (* DRIVE IN 'Switch on disabled' STATE *)
 	gpAx[nHliAxisIdx]^.lr_mc_control.drive_on.command_w				:= TRUE;
 
	IF wDriveState.0 THEN
		nState			:= 20; 
	ELSIF fbTonTimeOut.Q THEN
		bError			:= TRUE;
		nErrorId		:= ERR_TIME_OUT;
		nErrorState		:= nState;
		nState			:= 0;
	END_IF
	
(* -----------------------------------------------------------------------------------	*)
 20: (* DRIVE IN 'Ready to switch on' STATE *)
 	gpAx[nHliAxisIdx]^.lr_mc_control.torque_permission.command_w	:= TRUE;
	
	IF wDriveState.1 THEN
		nState			:= 30; 
	ELSIF fbTonTimeOut.Q THEN
		bError			:= TRUE;
		nErrorId		:= ERR_TIME_OUT;
		nErrorState		:= nState;
		nState			:= 0;
	END_IF
	
 (* -----------------------------------------------------------------------------------	*)
 30: (* DRIVE IN 'Switched on' STATE *)
 	gpAx[nHliAxisIdx]^.lr_mc_control.release_feedhold.command_w		:= TRUE;
	
	IF wDriveState.2 THEN
		nState			:= 40; 
	ELSIF fbTonTimeOut.Q THEN
		bError			:= TRUE;
		nErrorId		:= ERR_TIME_OUT;
		nErrorState		:= nState;
		nState			:= 0;
	END_IF
	
 (* -----------------------------------------------------------------------------------	*)
 40: (* DRIVE IN 'Operation enabled' STATE *)
	AC_ClearError();
	
END_CASE
END_ACTION

ACTION AC_ClearError:
THIS^.bError		:= FALSE;
THIS^.nErrorId		:= 0;
THIS^.nErrorState	:= 0;
END_ACTION

ACTION AC_ProfiDrive:
(* ProfiNet Drives are supported by the torque permission and Drive On  *)
gpAx[nHliAxisIdx]^.lr_mc_control.torque_permission.command_w	:= TRUE;
gpAx[nHliAxisIdx]^.lr_mc_control.drive_on.command_w				:= bEnable;
END_ACTION

ACTION AC_SercosDrive:
(****************************************************************************************)
(*										Status data										*)
(****************************************************************************************)
(* Ready state is derived from status word bit 15!										*)
bAxisIsReady	:= bReadyForControlLoopOn; 
 
(* Enabled state is derived from status word bits 14 and 15. IMPORTANT: In order to 	*)
(* take status word bit 03 into account  - which represents the time needed for 		*)
(* releasing the brake - axis specific parameter 'antr.sercos.evaluate_drive_follows_	*)
(* cmd' has to be set!!!																*) 
bAxisIsEnabled	:= bReadyForControlLoopOn AND bReadyForPowerOn;
 
(****************************************************************************************)
(*										Command data									*)
(****************************************************************************************)
(* ControlBit no. 14 is set statically in order to provide torque supported stopping of	*)
(* in case someone disables the axis during movement!									*) 
gpAx[nHliAxisIdx]^.lr_mc_control.torque_permission.command_w	:= TRUE;

(* Only control bits 13 and 15 are being (re-)set in order to achieve axis enabling!	*)
gpAx[nHliAxisIdx]^.lr_mc_control.release_feedhold.command_w		:= bEnable;
gpAx[nHliAxisIdx]^.lr_mc_control.drive_on.command_w				:= bEnable;
END_ACTION

ACTION AC_TerminalDrive:
(****************************************************************************************)
(*										Status data										*)
(****************************************************************************************)
(* Since there is no feedback available on the HLI axis enabled state wiöö be emulated!	*)
bAxisIsEnabled	:= bEnable;
bAxisIsReady	:= FALSE;
 
(****************************************************************************************)
(*										Command data									*)
(****************************************************************************************)
(* Terminal drives are supported by the torque permission control unit only!			*)
gpAx[nHliAxisIdx]^.lr_mc_control.torque_permission.command_w	:= bEnable;
gpAx[nHliAxisIdx]^.lr_mc_control.release_feedhold.command_w		:= FALSE;
gpAx[nHliAxisIdx]^.lr_mc_control.drive_on.command_w				:= FALSE;
END_ACTION

END_FUNCTION_BLOCK

// CNC/3 Control/HLI3_SetAxisReferenceOffset
FUNCTION_BLOCK HLI3_SetAxisReferenceOffset
VAR_INPUT
	Execute: BOOL;
	nHliAxisIdx: INT;
	nOffset:	LREAL;  (* Offset in mm *)
END_VAR
VAR_OUTPUT
	Busy  : BOOL;
	Done: BOOL;
	Error : BOOL;
	ErrorId : INT;
END_VAR
VAR
	nState : int;
	trigStart: R_TRIG;
END_VAR

(* ========================================================= *)
(*    FUN: HLI3_SetAxisReferenceOffset                      *)
(* --------------------------------------------------------- *)
(*   
    Desc: 
	Set reference offset position of an axis.
 
	To use this FB to set the offset for absolute encoder axis the following axis parameter settings should be done:
	
	kenngr.abs_pos_gueltig	0			( P-AXIS-00014 : Identification code for absolute path measurement system
	kenngr.set_refpos_mode	PLC_OFFSET  ( P-AXIS-00278 : Modes for setting the homing position (ABSOLUT / OFFSET /  PLC / PLC_OFFSET)
	
	While commanding the axis must not be involved in active interpolation or active manual mode!
	
	Errors:
	1 : nHliAxisIdx is invalid
*)
(*                                               
   Author: MiB                                               
   Date: 13.07.2017                                        
   Rev.: 1.0                                               
 =========================================================*) 
 
 trigStart(clk := Execute);
 IF trigStart.Q THEN  // start on flank of Execute
		 nState := 10;    
		 Done := FALSE;
		 Error := FALSE;
		 ErrorId := 0;
		 Busy := TRUE;
		gpAx[nHliAxisIdx]^.lr_mc_control.set_reference_position.command_w := FALSE;	 
		gpAx[nHliAxisIdx]^.lr_mc_control.clear_reference_position.command_w := FALSE;
 END_IF
 
 CASE nState OF
	 0: (* Idle *)
	 	Done := TRUE;
		Busy := FALSE;
	10: (* check Axis id valid *)
		IF NOT HLI3_CheckAxisValid(nHliAxisIdx := nHliAxisIdx) THEN	
			nState :=-1;
			Done := TRUE;
			Busy := FALSE;
			Error := TRUE;
			ErrorId := 1;		
		ELSE
			nState := nState + 10;		
		END_IF		
	20: (* Start *)
		(* set reference position *)
		gpAx[nHliAxisIdx]^.lr_mc_control.clear_reference_position.enable_w := TRUE;
		gpAx[nHliAxisIdx]^.lr_mc_control.clear_reference_position.command_w := TRUE;
		IF gpAx[nHliAxisIdx]^.lr_mc_control.clear_reference_position.state_r THEN
			gpAx[nHliAxisIdx]^.lr_mc_control.clear_reference_position.command_w := FALSE;
			nState := nState + 10;
		END_IF

	30: (* transfer new offset value *)
		gpAx[nHliAxisIdx]^.lr_mc_control.refpos_position.command_w := LREAL_TO_DINT(nOffset *10000.0);
		IF (gpAx[nHliAxisIdx]^.lr_mc_control.refpos_position.state_r = LREAL_TO_DINT(nOffset * 10000.0) ) THEN
			gpAx[nHliAxisIdx]^.lr_mc_control.set_reference_position.command_w := TRUE;
			nState := nState + 10;		
		END_IF
	40: (* tigger "write offset" *)
		
		IF (gpAx[nHliAxisIdx]^.lr_mc_control.set_reference_position.state_r) THEN
			gpAx[nHliAxisIdx]^.lr_mc_control.set_reference_position.command_w := FALSE;
			nState := 0;
		END_IF
	
	
 END_CASE

END_FUNCTION_BLOCK

// CNC/3 Control/HLI3_ClearReferencePosition
FUNCTION HLI3_ClearReferencePosition : BOOL
VAR_INPUT
	bExecute: BOOL;
	nHliAxisIdx: INT;
END_VAR

(* ========================================================= *)
(*    FUN: HLI3_ClearReferencePosition                       *)
(* --------------------------------------------------------- *)
(*   Desc:                                                   *)
(* 	 Author: TV                                              *)
(*   Date: 17.06.2015                                        *)
(*   Rev.: 1.0                                               *)
(* ========================================================= *)
HLI3_ClearReferencePosition := FALSE;

IF NOT HLI3_CheckAxisValid(nHliAxisIdx := nHliAxisIdx) THEN	
	RETURN;
END_IF

(* set reference position *)
gpAx[nHliAxisIdx]^.lr_mc_control.clear_reference_position.enable_w := TRUE;
gpAx[nHliAxisIdx]^.lr_mc_control.clear_reference_position.command_w := bExecute;
HLI3_ClearReferencePosition := TRUE;

END_FUNCTION

// CNC/3 Control/HLI3_SetProbingSignal
FUNCTION HLI3_SetProbingSignal : BOOL
VAR_INPUT
	nHliAxisIdx: INT;
	bProbingSignal: BOOL;
END_VAR


IF NOT HLI3_CheckAxisValid(nHliAxisIdx := nHliAxisIdx) THEN	
	HLI3_SetProbingSignal := FALSE;
	RETURN;
END_IF


gpAx[nHliAxisIdx]^.lr_mc_control.probing_signal.enable_w  := TRUE;
gpAx[nHliAxisIdx]^.lr_mc_control.probing_signal.command_w := bProbingSignal;
HLI3_SetProbingSignal := TRUE;

END_FUNCTION

// CNC/12 CNC_Axis/FB_ReadSWLimitSwitches
//*********************************************************************************************************
///NAME.......................:		FB_ReadSWLimitSwitches
///DATUM....................:		03.01.2018
///AUTOR....................:		Thomas Voß
///VERSION................:			1.1
///
///Description.: 	Read Software Limit Switches					
///**********************************************************************************************************

FUNCTION_BLOCK FB_ReadSWLimitSwitches
VAR_INPUT	
	nLogAxisNo		: UINT;		
	bExecute		: BOOL;
END_VAR
VAR_OUTPUT
	bError : BOOL;
	bBusy: BOOL;
	fSWLimitNeg		: LREAL;	(* Unit mm *)
	fSWLimitPos		: LREAL;	(* Unit mm *)
END_VAR
VAR
		fbOnTrigger		:  	R_TRIG;
		FbAdsRead		: 	ADSREAD;
		Step 			: 	UDINT;
		TimeOut 		: 	TON;	
		nSWLimitNeg 	: 	DINT;
		nSWLimitPos  	: 	DINT;
END_VAR

fbOnTrigger(CLK:= bExecute);


IF fbOnTrigger.Q THEN
	Step 	:= 10;	
	bError	:= 0;
	bBusy 	:= TRUE;
	FbAdsRead(READ := FALSE);
	
	fSWLimitNeg		:= 0;
	fSWLimitPos		:= 0;
	nSWLimitNeg 	:= 0;
	nSWLimitPos  	:= 0;
END_IF

CASE Step OF
0:
	bBusy 	:= FALSE;
	
10: (* Read negative Limit Switch *)

	IF nLogAxisNo < 1 OR  nLogAxisNo > MAX_SYS_LOG_AXIS_INDEX THEN
		Step := 999;
	ELSIF CNCSystem.LogAxisNo[nLogAxisNo].nHliAxisIdx = -1 THEN
		Step := 999;
	ELSE
		TimeOut(IN:=FALSE);
		FbAdsRead(	NETID:= '',							(* local *)
					PORT:= 553,							(* Port number of Task COM, all ADS-Requests to the NC-kernel  *)                          
					IDXGRP:=16#00020200+nLogAxisNo,    	(*  *)
					IDXOFFS:= 16#26,
					LEN:=SIZEOF(nSWLimitNeg),		(* number of bytes that shall be read                          *)
					DESTADDR:= ADR(nSWLimitNeg),  	(* memory for the read value, must be provided by the user     *)
					READ:=TRUE,							(* a rising edge on this input starts the read request         *)
					TMOUT:= T#1S);       				(* maximum time for read request                               *)
	
			Step := Step+10;
	END_IF

20:
		TimeOut(IN:=TRUE, PT:=T#2S);
		FbAdsRead();
		IF NOT FbAdsRead.Busy THEN
			IF NOT FbAdsRead.ERR THEN
				FbAdsRead(READ := FALSE);				
				fSWLimitNeg	 := DINT_TO_LREAL(nSWLimitNeg) / 10000.0; 				
				Step := Step+10;
			ELSE
				FbAdsRead(READ := FALSE);				
				Step := 999;
			END_IF
		END_IF

		(* error timeout *)
		IF TimeOut.Q THEN			
			Step   	:= 999;
		END_IF

30: (* Read positive Limit Switch *)
	TimeOut(IN:=FALSE);
	FbAdsRead(	NETID:= '',							(* local *)
				PORT:= 553,							(* Port number of Task COM, all ADS-Requests to the NC-kernel  *)
				IDXGRP:=16#00020200+nLogAxisNo,     (*  *)
				IDXOFFS:= 16#25,
				LEN:=SIZEOF(nSWLimitPos),		(* number of bytes that shall be read                          *)
				DESTADDR:= ADR(nSWLimitPos),  	(* memory for the read value, must be provided by the user     *)
				READ:=TRUE,							(* a rising edge on this input starts the read request         *)
				TMOUT:= T#1S);       				(* maximum time for read request                               *)
				
				Step := Step+10;

40:	TimeOut(IN:=TRUE, PT:=T#2S);
		FbAdsRead();
		IF NOT FbAdsRead.Busy THEN
			IF NOT FbAdsRead.ERR THEN
				FbAdsRead(READ := FALSE);
				fSWLimitPos	 := DINT_TO_LREAL(nSWLimitPos) / 10000.0;
				Step := 0;
			ELSE
				FbAdsRead(READ := FALSE);				
				Step := 999;
			END_IF
		END_IF
		
		(* error timeout *)
		IF TimeOut.Q THEN			
			Step   	:= 999;
		END_IF

		
999:	(* Error *)
		bError := TRUE;
		Step := 0;	
	
END_CASE

END_FUNCTION_BLOCK

// CNC/12 CNC_Axis/HLI3_CNCAxis
FUNCTION_BLOCK HLI3_CNCAxis EXTENDS HLI3_CNCAxisBase
VAR_INPUT
	nHliAxisIdx : INT := -1;
END_VAR
VAR_OUTPUT
END_VAR
VAR
END_VAR

(* ========================================================= *)
(*     FB: HLI3_CNCAxis                                  	 *)
(* --------------------------------------------------------- *)
(*   Desc:  CNC Axis Control							   	 *)
(*   Author: TV				                                 *)
(*   Date: 2018.01.25                                        *)
(*   Rev.: 1.0                                               *)
(* ==========================================================*)

SUPER^(nHliIdx := nHliAxisIdx);

END_FUNCTION_BLOCK

// CNC/13 Spindle/HLI3_HandleSpindleTechno
FUNCTION_BLOCK HLI3_HandleSpindleTechno
VAR_INPUT
	/// Logical axis number of the plc spindle 
	nHliAxisIdx: INT;
	/// The channel which commands the spindle, only used if 'bIsChannelSpecific' set TRUE 
	nHliChannelIdx: INT;
	/// Has to be set TRUE if the spindel intechno function is transmitted via the channel specific section of the HLI
	bIsChannelSpecific: BOOL;
	/// if using a plc controlled spindle: configured log_ax_nr in channel list 
	nLogAxisNoChannelSpecific: INT;
	/// Has to be set TRUE if zthis FB should car about gear change M functions M40 - M45
	bHandleGearChange: BOOL;
	/// Resets all internal states and variables of this function block 
	bChannelReset: BOOL;
END_VAR
VAR_OUTPUT
	/// Returns the commanded revolution programmed with a M03 or M05 [] 
	nRevolution: DINT;
	/// Returns the target position programmed with a M19 [0.1µm] or [] 
	nPosition: DINT;
	/// Error flag 
	bError: BOOL;
	/// Error id 
	nErrorId: UDINT;
END_VAR
VAR_IN_OUT
	/// Raises if the cnc program encounters a M03 for the relevant spindle. Reset this for acknowledge 
	M03: BOOL;
	/// Raises if the cnc program encounters a M04 for the relevant spindle. Reset this for acknowledge 
	M04: BOOL;
	/// Raises if the cnc program encounters a M05 for the relevant spindle. Reset this for acknowledge 
	M05: BOOL;
	/// Raises if the cnc program encounters a M19 for the relevant spindle. Reset this for acknowledge 
	M19: BOOL;
END_VAR
VAR
	/// Raises if the cnc program encounters a M40 for the relevant spindle. Reset this for acknowledge 
	pM40: POINTER TO BOOL;
	/// Raises if the cnc program encounters a M41 for the relevant spindle. Reset this for acknowledge 
	pM41: POINTER TO BOOL;
	/// Raises if the cnc program encounters a M42 for the relevant spindle. Reset this for acknowledge 
	pM42: POINTER TO BOOL;
	/// Raises if the cnc program encounters a M43 for the relevant spindle. Reset this for acknowledge 
	pM43: POINTER TO BOOL;
	/// Raises if the cnc program encounters a M44 for the relevant spindle. Reset this for acknowledge 
	pM44: POINTER TO BOOL;
	/// Raises if the cnc program encounters a M45 for the relevant spindle. Reset this for acknowledge 
	pM45: POINTER TO BOOL;	


	/// Number of open technology functions 
	nOpenTechnoCount: UINT;
	nOpenTechnoCountLate: UINT;
	
	/// Internal acknowledge signal 
	bAcknowledge: BOOL;
	/// Internal state of M03 request 
	M03_Internal: BOOL;
	/// Internal state of M04 request 
	M04_Internal: BOOL;
	/// Internal state of M05 request 
	M05_Internal: BOOL;
	/// Internal state of M19 request 
	M19_Internal: BOOL;
	/// Internal state of M19 request 
	M40_Internal: BOOL;
	/// Internal state of M19 request 
	M41_Internal: BOOL;
	/// Internal state of M19 request 
	M42_Internal: BOOL;
	/// Internal state of M19 request 
	M43_Internal: BOOL;
	/// Internal state of M19 request 
	M44_Internal: BOOL;
	/// Internal state of M19 request 
	M45_Internal: BOOL;
	/// Index of axis specific HLI area 
	nHliAxIfcIdx: UDINT;
	/// Index of axis specific technology function at HLI 
	nTechFctMaxIdx: UINT;
	nTechFctMaxIdxLate: UINT;
	/// Counting variable for loop processing 
	nLoop: UINT;
	
	/// Pointer to spindle specific data 
	pSProcess: POINTER TO HLI_S_PROZESS;
	pMProcess: POINTER TO HLI_M_H_PROZESS;
	/// Rising trigger of input 'bChannelReset' 
	fbRtrigChannelReset: R_TRIG;
	
	bFirstRun : BOOL := TRUE;
	dummyM40: BOOL;
	dummyM41: BOOL;
	dummyM42: BOOL;
	dummyM43: BOOL;
	dummyM44: BOOL;
	dummyM45: BOOL;
	
END_VAR

(****************************************************************************************)
(* POU:		HLI3_HandlePlcSpindle                      									*)
(* Type:	Function Block																*)
(* Author: 	HR, MiB, TV																    *)
(* Date: 	10/11/10																	*)
(* Rev.: 	1.0																			*)
(* Rev.: 	1.6	14/10/23    															*)
(* ------------------------------------------------------------------------------------ *)
(* Desc:	Function block for handling technology functions of PLC spindles. It works	*)
(*			properly if there is a ation axis in the configuration. The logical 		*)
(*			axis no. 'n' of that axis is used to indetify that spindle in this function	*)
(*			block. This implies a spindle configuration like the folowing:				*)
(*				spdl_anzahl                         1	(maybe more?)					*)
(*				main_spindle_ax_nr                  n	(enter right value there)		*)
(*				main_spindle_name                   S									*)
(*				spindle_m_fct_free                  0									*)
(*				spindel[0].bezeichnung              S1									*)
(*				spindel[0].log_achs_nr              n	(enter right value there)		*)
(*				spindel[0].plc_control              1									*)
(*																						*)
(*			The function block may raise some errors specified by an error id:			*)
(*				+ 10000: axis number not valid!											*)
(*																						*)
(****************************************************************************************)
(* Date:	13/09/16																	*)
(* Author:	RCH																			*)
(* Rev:		1.1																			*)
(* ------------------------------------------------------------------------------------ *)
(* Desc 	Renamed, according to Tc2 version. This FB also works for CNC spindles with	*) 
(*			S or M functions set to inform PLC. 										*)
(****************************************************************************************)
(* Date:	13/09/16																	*)
(* Author:	RCH																			*)
(* Rev:		1.2																			*)
(* ------------------------------------------------------------------------------------ *)
(* Desc 	Introduced new input parameters 'bIsChannelSpecific' and 'nChannelNo' in 	*)
(*			order to make this FB work for PLC spindles which are sending synch.		*)
(*			requests via the channel specific section of the HLI. Here the spindle		*)
(* 			specific parameters have to be set as follows:								*)
(*				spindel[n].plc_control            1			(P-CHAN-00069)				*)
(*				spindel[n].log_achs_nr            m			(P-CHAN-00036)				*)
(*																						*)
(*			The logical axis number in P-CHAN-00036 used for such a spindle must not be	*)
(*			lower than one and must not be used by any other axis. This FB works if the	*)
(*			value of this logical axis number fits the parameter 'nHliAxisIdx' only!	*)
(* 																						*)
(*			In order to guarantee save HLI access the following new error codes have	*)
(*			been introduced:															*)
(*				+ 20000: Channel no lower than one!										*)
(*				+ 20001: Channel number exceeds number of configured channels.			*)
(*				+ 20002: No HLI data for channel.										*)
(****************************************************************************************)
(* Date:	14/01/22																	*)
(* Author:	TV																			*)
(* Rev:		1.3																			*)
(* ------------------------------------------------------------------------------------ *)
(* Desc:	bugfix in function to check nHLIAxisIdx and LogAxisId						*) 
(****************************************************************************************)
(* Date:	14/09/10																	*)
(* Author:	RCH																			*)
(* Rev:		1.4																			*)
(* ------------------------------------------------------------------------------------ *)
(* Desc 	Added optional handling of spindle gear change M functions M40 - M45.		*)
(****************************************************************************************)
(* Date:	14/09/12																	*)
(* Author:	RCH																			*)
(* Rev:		1.5																			*)
(* ------------------------------------------------------------------------------------ *)
(* Desc 	Fixed bug with spindle M functions send by the channel spec. section of the	*)
(*			HLI. So far the channel specific section was used for determining the value *)
(*			of  'nTechFctMaxidx'.														*)
(****************************************************************************************)
(* Date:	14/10/23																	*)
(* Author:	MiB																			*)
(* Rev:		1.6																			*)
(* ------------------------------------------------------------------------------------ *)
(* Desc 	Introduced parameter "nLogAxisNoChannelSpecific" which allows to use a plc  *)
(*			spindle without a simulation axis for the spindle. 				 			*)
(*			This paramater is only used if "bIsChannelSpecific == true"					*)
(*																						*)
(*				spindel[n].plc_control            1			(P-CHAN-00069)				*)
(*				spindel[n].log_achs_nr            m			(P-CHAN-00036)				*)
(*																						*)
(*			The logical axis number in P-CHAN-00036 used for such a spindle must not be	*)
(*			lower than one and must not be used by any other axis. This FB works if the	*)
(*			value of this logical axis number fits the parameter 						*)
(*			'nLogAxisNoChannelSpecific' only!											*)
(****************************************************************************************)
(* Date:	15/03/05																	*)
(* Author:	MiB																			*)
(* Rev:		1.7																			*)
(* ------------------------------------------------------------------------------------ *)
(* Desc 	Removed gearchange m functions from var_in_out							    *)
(*			Created new FB HLI3_SpindleTechnoGearchange									*)
(****************************************************************************************)
(*								Init Pointer to pM40..pM45								*)
(****************************************************************************************)
(* Date:	17/02/03																	*)
(* Author:	MiB																			*)
(* Rev:		1.7																			*)
(* ------------------------------------------------------------------------------------ *)
(* Desc 	Handling of late sync M functions. 											*)
(*			Usage of different structure TECHNO_UNIT_AX and TECHNO_UNIT_CH, depending 	*)
(*			on channel or axis specific specific interface 							 	*)
(****************************************************************************************)
(* Date:	19/04/19																	*)
(* Author:	TV																			*)
(* Rev:		1.8																			*)
(* ------------------------------------------------------------------------------------ *)
(* Desc 	Reset the M-Function flags after Reset										*)
(****************************************************************************************)


IF bFirstRun THEN
	bFirstRun := FALSE;
	pM40 := ADR(dummyM40);
	pM41 := ADR(dummyM41);
	pM42 := ADR(dummyM42);
	pM43 := ADR(dummyM43);
	pM44 := ADR(dummyM44);
	pM45 := ADR(dummyM45);	
END_IF

A_HandleTechno();

ACTION A_HandleTechno:

(****************************************************************************************)
(*								Cyclic reset of  error flag 							*)
(****************************************************************************************)
bError										:= FALSE;
nErrorId									:= 0;

(****************************************************************************************)
(*							  Check for valid logical axis no.							*)
(****************************************************************************************)
IF NOT bIsChannelSpecific AND NOT HLI3_CheckAxisValid(nHliAxisIdx := nHliAxisIdx) THEN
	bError									:= TRUE;
	nErrorId								:= 10000;
	RETURN;
END_IF

IF NOT HLI3_CheckChannelValid(nChannel := nHliChannelIdx) THEN
	bError									:= TRUE;
	nErrorId								:= 20000;
	RETURN;	
END_IF

(****************************************************************************************)
(*											Reset										*)
(****************************************************************************************)
fbRtrigChannelReset
	(CLK := bChannelReset);

IF fbRtrigChannelReset.Q THEN
	M_Reset(M03:=M03, M04:=M04,M05:=M05,M19:=M19);
END_IF

(****************************************************************************************)
(*									Receive requests from cnc							*)
(****************************************************************************************)
(* Look out for open technology function either on the channel or the axis specific		*)
(* section of the HLI, depending on parameter ''.										*)
IF bIsChannelSpecific THEN
	nOpenTechnoCount	:= gpCh[nHliChannelIdx]^.used_units_std_sync_r;
	nOpenTechnoCountLate:= gpCh[nHliChannelIdx]^.used_units_late_sync_r;
	
